C07189=1022.011,-71.493,-94.373,166.291,49.653,158.986
C07190=1022.017,-71.243,-94.384,166.295,49.649,158.986
C07191=1022.023,-70.994,-94.395,166.298,49.645,158.986
C07192=1022.028,-70.744,-94.405,166.301,49.641,158.985
C07193=1022.034,-70.494,-94.416,166.303,49.637,158.985
C07194=1022.040,-70.245,-94.427,166.306,49.634,158.985
C07195=1022.045,-69.995,-94.438,166.309,49.630,158.985
C07196=1022.051,-69.745,-94.448,166.312,49.627,158.985
C07197=1022.057,-69.465,-94.461,166.316,49.622,158.984
C07198=1022.063,-69.184,-94.472,166.319,49.618,158.984
C07199=1022.070,-68.903,-94.485,166.322,49.613,158.984
C07200=1022.076,-68.622,-94.497,166.326,49.609,158.984
C07201=1022.082,-68.373,-94.507,166.329,49.606,158.984
C07202=1022.087,-68.123,-94.518,166.332,49.601,158.983
C07203=1022.093,-67.874,-94.529,166.335,49.598,158.983
C07204=1022.099,-67.624,-94.540,166.338,49.594,158.983
C07205=1022.104,-67.374,-94.550,166.340,49.590,158.983
C07206=1022.110,-67.125,-94.561,166.343,49.587,158.983
C07207=1022.115,-66.875,-94.573,166.347,49.582,158.982
C07208=1022.121,-66.626,-94.583,166.350,49.578,158.982
C07209=1022.127,-66.376,-94.594,166.353,49.575,158.982
C07210=1022.132,-66.127,-94.605,166.356,49.571,158.982
C07211=1022.138,-65.876,-94.616,166.359,49.567,158.981
C07212=1022.144,-65.626,-94.627,166.362,49.564,158.981
C07213=1022.150,-65.377,-94.637,166.364,49.560,158.981
C07214=1022.156,-65.127,-94.648,166.368,49.555,158.981
C07215=1022.161,-64.878,-94.659,166.371,49.552,158.981
C07216=1022.166,-64.628,-94.671,166.374,49.548,158.980
C07217=1022.172,-64.378,-94.682,166.377,49.544,158.980
C07218=1022.178,-64.128,-94.693,166.379,49.540,158.980
C07219=1022.184,-63.879,-94.704,166.383,49.537,158.980
C07220=1022.190,-63.629,-94.714,166.385,49.533,158.979
C07221=1022.195,-63.379,-94.725,166.388,49.529,158.979
C07222=1022.201,-63.130,-94.736,166.392,49.525,158.979
C07223=1022.207,-62.880,-94.746,166.395,49.521,158.979
C07224=1022.213,-62.630,-94.758,166.398,49.517,158.979
C07225=1022.218,-62.380,-94.769,166.400,49.513,158.978
C07226=1022.224,-62.131,-94.780,166.404,49.510,158.978
C07227=1022.230,-61.881,-94.791,166.406,49.506,158.978
C07228=1022.236,-61.631,-94.802,166.409,49.502,158.978
C07229=1022.242,-61.382,-94.813,166.413,49.498,158.978
C07230=1022.247,-61.132,-94.824,166.416,49.494,158.977
C07231=1022.253,-60.883,-94.835,166.419,49.490,158.977
///RCONF 1,0,0,0,0,0,0,0,0,0,0,0,0,0,0,0,0,0,0,0,0,0,0,0
C07232=1022.259,-60.633,-94.846,166.421,49.486,158.977
C07233=1022.264,-60.383,-94.858,166.424,49.482,158.977
C07234=1022.270,-60.133,-94.868,166.427,49.479,158.976
C07235=1022.276,-59.884,-94.879,166.431,49.474,158.976
C07236=1022.282,-59.634,-94.890,166.434,49.470,158.976
C07237=1022.288,-59.385,-94.902,166.437,49.466,158.976
C07238=1022.294,-59.135,-94.913,166.440,49.463,158.976
C07239=1022.300,-58.886,-94.924,166.442,49.459,158.975
C07240=1022.305,-58.635,-94.936,166.445,49.455,158.975
C07241=1022.311,-58.386,-94.947,166.448,49.451,158.975
C07242=1022.317,-58.136,-94.957,166.452,49.447,158.975
C07243=1022.323,-57.887,-94.968,166.455,49.443,158.974
C07244=1022.329,-57.636,-94.980,166.458,49.439,158.974
C07245=1022.335,-57.387,-94.990,166.460,49.435,158.974
C07246=1022.340,-57.137,-95.001,166.463,49.431,158.974
C07247=1022.346,-56.888,-95.014,166.466,49.427,158.973
C07248=1022.352,-56.638,-95.025,166.470,49.424,158.973
C07249=1022.358,-56.389,-95.036,166.473,49.420,158.973
C07250=1022.364,-56.138,-95.047,166.475,49.416,158.973
C07251=1022.370,-55.889,-95.058,166.478,49.412,158.972
C07252=1022.376,-55.639,-95.069,166.481,49.408,158.972
C07253=1022.382,-55.390,-95.081,166.484,49.404,158.972
C07254=1022.387,-55.140,-95.092,166.488,49.400,158.972
C07255=1022.394,-54.890,-95.103,166.491,49.396,158.971
C07256=1022.399,-54.640,-95.114,166.493,49.392,158.971
C07257=1022.405,-54.391,-95.125,166.496,49.388,158.971
C07258=1022.412,-54.141,-95.137,166.499,49.384,158.971
C07259=1022.418,-53.892,-95.148,166.502,49.380,158.970
C07260=1022.423,-53.641,-95.160,166.505,49.376,158.970
C07261=1022.430,-53.363,-95.172,166.508,49.372,158.970
C07262=1022.437,-53.083,-95.185,166.512,49.367,158.970
C07263=1022.443,-52.803,-95.197,166.515,49.362,158.969
C07264=1022.450,-52.524,-95.210,166.518,49.358,158.969
C07265=1022.456,-52.274,-95.221,166.521,49.354,158.969
C07266=1022.462,-52.025,-95.233,166.525,49.350,158.969
C07267=1022.467,-51.775,-95.244,166.527,49.346,158.968
C07268=1022.474,-51.525,-95.256,166.530,49.342,158.968
C07269=1022.480,-51.276,-95.267,166.533,49.338,158.968
C07270=1022.485,-51.026,-95.278,166.536,49.335,158.968
C07271=1022.492,-50.776,-95.289,166.540,49.330,158.967
C07272=1022.497,-50.527,-95.302,166.543,49.326,158.967
C07273=1022.503,-50.276,-95.313,166.545,49.322,158.967
C07274=1022.509,-50.028,-95.325,166.548,49.319,158.967
C07275=1022.514,-49.777,-95.337,166.551,49.315,158.966
C07276=1022.520,-49.528,-95.348,166.554,49.312,158.966
C07277=1022.526,-49.278,-95.360,166.557,49.308,158.966
C07278=1022.532,-49.029,-95.372,166.560,49.304,158.966
C07279=1022.538,-48.778,-95.384,166.563,49.300,158.966
C07280=1022.544,-48.529,-95.395,166.566,49.296,158.965
C07281=1022.550,-48.279,-95.408,166.568,49.292,158.965
C07282=1022.555,-48.030,-95.419,166.572,49.289,158.965
C07283=1022.561,-47.780,-95.431,166.574,49.285,158.965
C07284=1022.566,-47.530,-95.443,166.577,49.281,158.964
C07285=1022.573,-47.281,-95.455,166.580,49.277,158.964
C07286=1022.578,-47.031,-95.466,166.583,49.274,158.964
C07287=1022.585,-46.781,-95.478,166.586,49.270,158.964
C07288=1022.590,-46.532,-95.490,166.588,49.266,158.963
C07289=1022.596,-46.282,-95.502,166.592,49.263,158.963
C07290=1022.601,-46.033,-95.514,166.594,49.259,158.963
C07291=1022.607,-45.783,-95.526,166.598,49.254,158.963
C07292=1022.613,-45.533,-95.537,166.601,49.251,158.963
C07293=1022.619,-45.284,-95.550,166.604,49.247,158.962
C07294=1022.625,-45.035,-95.561,166.607,49.243,158.962
C07295=1022.631,-44.784,-95.573,166.610,49.239,158.962
C07296=1022.636,-44.535,-95.585,166.613,49.236,158.962
C07297=1022.643,-44.285,-95.597,166.615,49.232,158.961
C07298=1022.648,-44.035,-95.609,166.618,49.228,158.961
C07299=1022.654,-43.786,-95.621,166.621,49.224,158.961
C07300=1022.660,-43.536,-95.633,166.624,49.221,158.961
C07301=1022.666,-43.287,-95.644,166.627,49.217,158.960
C07302=1022.672,-43.037,-95.657,166.630,49.213,158.960
C07303=1022.677,-42.788,-95.669,166.632,49.209,158.960
C07304=1022.684,-42.538,-95.681,166.635,49.205,158.960
C07305=1022.689,-42.288,-95.693,166.638,49.201,158.959
C07306=1022.695,-42.039,-95.704,166.642,49.197,158.959
C07307=1022.701,-41.789,-95.717,166.645,49.193,158.959
C07308=1022.707,-41.539,-95.729,166.648,49.189,158.958
C07309=1022.713,-41.289,-95.740,166.651,49.186,158.958
C07310=1022.719,-41.040,-95.753,166.653,49.182,158.958
C07311=1022.725,-40.791,-95.764,166.656,49.178,158.958
C07312=1022.731,-40.541,-95.777,166.659,49.174,158.957
C07313=1022.737,-40.291,-95.790,166.662,49.170,158.957
C07314=1022.743,-40.041,-95.800,166.665,49.167,158.957
C07315=1022.748,-39.792,-95.813,166.668,49.163,158.957
C07316=1022.755,-39.542,-95.825,166.670,49.159,158.956
C07317=1022.760,-39.293,-95.837,166.673,49.155,158.956
C07318=1022.766,-39.043,-95.850,166.676,49.151,158.956
C07319=1022.772,-38.793,-95.862,166.679,49.147,158.956
C07320=1022.779,-38.543,-95.874,166.682,49.143,158.955
C07321=1022.784,-38.294,-95.886,166.685,49.139,158.955
C07322=1022.790,-38.044,-95.899,166.688,49.136,158.955
C07323=1022.796,-37.794,-95.911,166.690,49.132,158.955
C07324=1022.801,-37.545,-95.923,166.693,49.128,158.954
C07325=1022.808,-37.266,-95.937,166.697,49.124,158.954
C07326=1022.815,-36.986,-95.951,166.700,49.120,158.954
C07327=1022.821,-36.708,-95.965,166.704,49.116,158.954
C07328=1022.828,-36.429,-95.979,166.706,49.112,158.953
C07329=1022.834,-36.179,-95.992,166.709,49.108,158.953
C07330=1022.839,-35.929,-96.004,166.712,49.104,158.953
C07331=1022.845,-35.680,-96.016,166.715,49.100,158.953
C07332=1022.851,-35.430,-96.028,166.718,49.096,158.952
C07333=1022.857,-35.180,-96.041,166.721,49.093,158.952
C07334=1022.863,-34.931,-96.053,166.724,49.089,158.952
C07335=1022.869,-34.681,-96.066,166.726,49.085,158.952
C07336=1022.875,-34.431,-96.078,166.729,49.081,158.951
C07337=1022.880,-34.181,-96.091,166.732,49.078,158.951
C07338=1022.886,-33.932,-96.103,166.735,49.074,158.951
C07339=1022.892,-33.682,-96.115,166.738,49.070,158.951
C07340=1022.898,-33.433,-96.127,166.741,49.066,158.950
C07341=1022.904,-33.183,-96.141,166.744,49.063,158.950
C07342=1022.910,-32.934,-96.153,166.747,49.059,158.950
C07343=1022.916,-32.684,-96.165,166.749,49.055,158.950
C07344=1022.922,-32.434,-96.178,166.752,49.051,158.949
C07345=1022.928,-32.185,-96.191,166.755,49.048,158.949
C07346=1022.933,-31.935,-96.203,166.758,49.044,158.949
C07347=1022.939,-31.686,-96.215,166.761,49.040,158.949
C07348=1022.945,-31.436,-96.229,166.764,49.036,158.948
C07349=1022.952,-31.187,-96.240,166.767,49.032,158.948
C07350=1022.958,-30.937,-96.253,166.769,49.028,158.948
C07351=1022.963,-30.687,-96.266,166.772,49.024,158.948
C07352=1022.969,-30.437,-96.278,166.775,49.020,158.947
C07353=1022.975,-30.188,-96.291,166.778,49.017,158.947
C07354=1022.981,-29.939,-96.304,166.781,49.013,158.947
C07355=1022.987,-29.689,-96.316,166.784,49.009,158.946
C07356=1022.993,-29.439,-96.329,166.786,49.005,158.946
C07357=1022.999,-29.189,-96.341,166.789,49.001,158.946
C07358=1023.006,-28.940,-96.354,166.792,48.997,158.946
C07359=1023.011,-28.690,-96.366,166.795,48.994,158.945
C07360=1023.017,-28.441,-96.379,166.798,48.990,158.945
C07361=1023.023,-28.192,-96.392,166.801,48.986,158.945
C07362=1023.029,-27.942,-96.405,166.804,48.982,158.945
C07363=1023.035,-27.692,-96.417,166.807,48.978,158.944
C07364=1023.041,-27.442,-96.430,166.810,48.974,158.944
C07365=1023.047,-27.193,-96.443,166.812,48.971,158.944
C07366=1023.053,-26.943,-96.455,166.815,48.967,158.943
C07367=1023.059,-26.694,-96.469,166.818,48.963,158.943
C07368=1023.064,-26.443,-96.482,166.821,48.960,158.943
C07369=1023.070,-26.194,-96.494,166.824,48.956,158.943
C07370=1023.076,-25.945,-96.507,166.826,48.952,158.942
C07371=1023.082,-25.695,-96.520,166.829,48.949,158.942
C07372=1023.088,-25.446,-96.533,166.832,48.945,158.942
C07373=1023.094,-25.196,-96.546,166.835,48.941,158.942
C07374=1023.099,-24.946,-96.560,166.838,48.938,158.942
C07375=1023.105,-24.696,-96.572,166.841,48.934,158.941
C07376=1023.111,-24.447,-96.585,166.844,48.930,158.941
C07377=1023.117,-24.197,-96.598,166.847,48.926,158.941
C07378=1023.123,-23.948,-96.611,166.850,48.922,158.941
C07379=1023.129,-23.698,-96.624,166.852,48.918,158.940
C07380=1023.135,-23.449,-96.638,166.854,48.915,158.940
C07381=1023.141,-23.199,-96.650,166.857,48.912,158.940
C07382=1023.147,-22.949,-96.663,166.860,48.908,158.939
C07383=1023.153,-22.700,-96.676,166.863,48.904,158.939
C07384=1023.159,-22.450,-96.689,166.866,48.900,158.939
C07385=1023.164,-22.200,-96.702,166.869,48.896,158.939
C07386=1023.170,-21.951,-96.716,166.871,48.892,158.938
C07387=1023.176,-21.701,-96.728,166.874,48.889,158.938
C07388=1023.183,-21.452,-96.742,166.877,48.885,158.938
C07389=1023.189,-21.172,-96.756,166.880,48.881,158.937
C07390=1023.196,-20.892,-96.771,166.884,48.876,158.937
C07391=1023.202,-20.612,-96.786,166.886,48.872,158.937
C07392=1023.209,-20.332,-96.800,166.890,48.867,158.937
C07393=1023.215,-20.083,-96.813,166.893,48.864,158.936
C07394=1023.221,-19.833,-96.826,166.896,48.860,158.936
C07395=1023.227,-19.582,-96.840,166.899,48.856,158.936
C07396=1023.233,-19.333,-96.853,166.901,48.852,158.935
C07397=1023.239,-19.084,-96.866,166.903,48.849,158.935
C07398=1023.245,-18.834,-96.879,166.906,48.845,158.935
C07399=1023.251,-18.585,-96.892,166.909,48.842,158.935
C07400=1023.257,-18.335,-96.906,166.912,48.838,158.934
C07401=1023.263,-18.085,-96.919,166.915,48.834,158.934
C07402=1023.269,-17.836,-96.932,166.917,48.830,158.934
C07403=1023.275,-17.587,-96.945,166.921,48.826,158.934
C07404=1023.281,-17.337,-96.958,166.923,48.822,158.933
C07405=1023.287,-17.087,-96.972,166.926,48.819,158.933
C07406=1023.293,-16.838,-96.985,166.929,48.815,158.933
C07407=1023.299,-16.588,-96.997,166.932,48.811,158.932
C07408=1023.305,-16.339,-97.011,166.934,48.807,158.932
C07409=1023.312,-16.089,-97.024,166.938,48.803,158.932
C07410=1023.317,-15.839,-97.038,166.940,48.800,158.932
C07411=1023.323,-15.589,-97.051,166.943,48.796,158.931
C07412=1023.329,-15.340,-97.064,166.946,48.792,158.931
C07413=1023.335,-15.091,-97.078,166.949,48.788,158.931
C07414=1023.341,-14.841,-97.091,166.951,48.785,158.930
C07415=1023.346,-14.592,-97.105,166.954,48.781,158.930
C07416=1023.353,-14.343,-97.118,166.956,48.777,158.930
C07417=1023.359,-14.092,-97.132,166.960,48.774,158.930
C07418=1023.365,-13.842,-97.145,166.962,48.770,158.929
C07419=1023.370,-13.593,-97.159,166.965,48.766,158.929
C07420=1023.376,-13.344,-97.172,166.968,48.763,158.929
C07421=1023.382,-13.094,-97.186,166.971,48.759,158.929
C07422=1023.388,-12.845,-97.199,166.973,48.755,158.928
C07423=1023.394,-12.595,-97.213,166.976,48.751,158.928
C07424=1023.400,-12.345,-97.227,166.979,48.748,158.928
C07425=1023.406,-12.096,-97.241,166.982,48.744,158.927
C07426=1023.412,-11.846,-97.254,166.984,48.740,158.927
C07427=1023.418,-11.597,-97.268,166.987,48.736,158.927
C07428=1023.424,-11.347,-97.281,166.990,48.733,158.927
C07429=1023.429,-11.098,-97.295,166.993,48.729,158.926
C07430=1023.436,-10.848,-97.309,166.996,48.725,158.926
C07431=1023.442,-10.598,-97.322,166.998,48.721,158.926
C07432=1023.448,-10.349,-97.336,167.001,48.718,158.925
C07433=1023.454,-10.100,-97.349,167.004,48.714,158.925
C07434=1023.459,-9.850,-97.363,167.006,48.710,158.925
C07435=1023.466,-9.600,-97.376,167.009,48.706,158.924
C07436=1023.472,-9.351,-97.390,167.012,48.703,158.924
C07437=1023.478,-9.101,-97.404,167.015,48.699,158.924
C07438=1023.483,-8.852,-97.417,167.018,48.695,158.924
C07439=1023.490,-8.602,-97.431,167.021,48.691,158.923
C07440=1023.496,-8.352,-97.445,167.022,48.687,158.923
C07441=1023.502,-8.103,-97.458,167.025,48.684,158.923
C07442=1023.507,-7.854,-97.472,167.028,48.680,158.923
C07443=1023.514,-7.604,-97.485,167.031,48.676,158.922
C07444=1023.520,-7.354,-97.500,167.034,48.672,158.922
C07445=1023.526,-7.105,-97.513,167.037,48.669,158.922
C07446=1023.531,-6.855,-97.527,167.039,48.665,158.921
C07447=1023.538,-6.605,-97.540,167.042,48.661,158.921
C07448=1023.544,-6.356,-97.555,167.045,48.657,158.921
C07449=1023.550,-6.107,-97.568,167.047,48.654,158.920
C07450=1023.556,-5.857,-97.582,167.050,48.650,158.920
C07451=1023.562,-5.607,-97.596,167.053,48.646,158.920
C07452=1023.568,-5.358,-97.610,167.056,48.642,158.919
C07453=1023.575,-5.076,-97.625,167.059,48.638,158.919
C07454=1023.582,-4.794,-97.641,167.062,48.633,158.919
C07455=1023.589,-4.513,-97.656,167.065,48.629,158.918
C07456=1023.596,-4.231,-97.671,167.069,48.625,158.918
C07457=1023.602,-3.981,-97.686,167.071,48.621,158.918
C07458=1023.607,-3.732,-97.700,167.073,48.618,158.917
C07459=1023.613,-3.483,-97.714,167.076,48.614,158.917
C07460=1023.619,-3.232,-97.728,167.079,48.610,158.917
C07461=1023.625,-2.983,-97.742,167.082,48.606,158.917
C07462=1023.631,-2.734,-97.756,167.085,48.603,158.917
C07463=1023.637,-2.484,-97.770,167.087,48.600,158.916
C07464=1023.643,-2.234,-97.784,167.090,48.596,158.916
C07465=1023.648,-1.985,-97.799,167.093,48.592,158.916
C07466=1023.654,-1.735,-97.813,167.095,48.589,158.915
C07467=1023.660,-1.486,-97.828,167.098,48.585,158.915
C07468=1023.666,-1.236,-97.842,167.100,48.582,158.915
C07469=1023.672,-0.986,-97.856,167.103,48.578,158.915
C07470=1023.678,-0.738,-97.870,167.106,48.574,158.914
C07471=1023.684,-0.488,-97.884,167.109,48.570,158.914
C07472=1023.690,-0.238,-97.899,167.112,48.567,158.914
C07473=1023.696,0.011,-97.912,167.114,48.563,158.913
C07474=1023.701,0.261,-97.926,167.116,48.559,158.913
C07475=1023.707,0.510,-97.941,167.120,48.556,158.913
C07476=1023.713,0.760,-97.955,167.122,48.552,158.913
C07477=1023.719,1.009,-97.969,167.125,48.548,158.912
C07478=1023.726,1.259,-97.983,167.127,48.545,158.912
C07479=1023.731,1.508,-97.998,167.130,48.541,158.912
C07480=1023.737,1.758,-98.012,167.133,48.537,158.911
C07481=1023.743,2.007,-98.027,167.136,48.533,158.911
C07482=1023.749,2.257,-98.041,167.139,48.530,158.911
C07483=1023.755,2.507,-98.055,167.141,48.527,158.910
C07484=1023.761,2.756,-98.069,167.143,48.523,158.910
C07485=1023.767,3.006,-98.083,167.146,48.519,158.910
C07486=1023.773,3.255,-98.098,167.149,48.515,158.909
C07487=1023.779,3.504,-98.112,167.152,48.512,158.909
C07488=1023.785,3.754,-98.126,167.154,48.508,158.909
C07489=1023.791,4.003,-98.141,167.157,48.504,158.909
C07490=1023.797,4.253,-98.155,167.160,48.500,158.908
C07491=1023.803,4.502,-98.170,167.162,48.496,158.908
C07492=1023.809,4.753,-98.184,167.166,48.493,158.908
C07493=1023.814,5.002,-98.199,167.167,48.489,158.907
C07494=1023.821,5.251,-98.212,167.170,48.486,158.907
C07495=1023.827,5.500,-98.227,167.173,48.482,158.907
C07496=1023.833,5.751,-98.241,167.176,48.478,158.906
C07497=1023.839,6.000,-98.256,167.179,48.474,158.906
C07498=1023.845,6.249,-98.271,167.182,48.471,158.906
C07499=1023.851,6.499,-98.284,167.183,48.467,158.906
C07500=1023.857,6.749,-98.299,167.186,48.463,158.905
C07501=1023.863,6.998,-98.313,167.189,48.459,158.905
C07502=1023.869,7.248,-98.328,167.192,48.455,158.905
C07503=1023.876,7.496,-98.342,167.195,48.451,158.904
C07504=1023.882,7.747,-98.356,167.197,48.449,158.904
C07505=1023.887,7.996,-98.371,167.200,48.445,158.904
C07506=1023.894,8.245,-98.386,167.202,48.441,158.903
C07507=1023.899,8.495,-98.400,167.205,48.437,158.903
C07508=1023.906,8.745,-98.415,167.208,48.433,158.903
C07509=1023.911,8.994,-98.429,167.211,48.429,158.902
C07510=1023.918,9.244,-98.444,167.213,48.425,158.902
C07511=1023.923,9.493,-98.458,167.215,48.421,158.902
C07512=1023.930,9.742,-98.473,167.218,48.418,158.901
C07513=1023.936,9.992,-98.486,167.221,48.414,158.901
C07514=1023.942,10.241,-98.501,167.224,48.410,158.901
C07515=1023.948,10.490,-98.516,167.227,48.407,158.901
C07516=1023.954,10.740,-98.531,167.229,48.403,158.900
C07517=1023.962,11.023,-98.547,167.232,48.398,158.900
C07518=1023.968,11.307,-98.564,167.235,48.394,158.899
C07519=1023.975,11.591,-98.581,167.238,48.390,158.899
C07520=1023.982,11.874,-98.597,167.242,48.385,158.899
C07521=1023.988,12.124,-98.611,167.244,48.382,158.898
C07522=1023.994,12.373,-98.626,167.247,48.378,158.898
C07523=1024.000,12.623,-98.641,167.249,48.374,158.898
C07524=1024.007,12.873,-98.656,167.252,48.370,158.897
C07525=1024.012,13.122,-98.670,167.255,48.366,158.897
C07526=1024.019,13.372,-98.684,167.257,48.362,158.897
C07527=1024.025,13.622,-98.699,167.260,48.358,158.896
C07528=1024.031,13.871,-98.714,167.262,48.356,158.896
C07529=1024.037,14.120,-98.729,167.265,48.352,158.896
C07530=1024.043,14.369,-98.743,167.268,48.348,158.895
C07531=1024.049,14.619,-98.758,167.271,48.344,158.895
C07532=1024.055,14.869,-98.774,167.273,48.340,158.895
C07533=1024.061,15.118,-98.789,167.276,48.337,158.895
C07534=1024.067,15.367,-98.803,167.278,48.333,158.894
C07535=1024.073,15.616,-98.818,167.281,48.329,158.894
C07536=1024.079,15.866,-98.833,167.284,48.325,158.894
C07537=1024.085,16.117,-98.848,167.286,48.322,158.893
C07538=1024.090,16.366,-98.862,167.289,48.319,158.893
C07539=1024.097,16.615,-98.877,167.292,48.315,158.893
C07540=1024.103,16.865,-98.892,167.295,48.311,158.892
C07541=1024.109,17.114,-98.907,167.296,48.307,158.892
C07542=1024.115,17.364,-98.922,167.299,48.303,158.892
C07543=1024.121,17.613,-98.937,167.302,48.299,158.891
C07544=1024.127,17.862,-98.952,167.305,48.296,158.891
C07545=1024.133,18.112,-98.967,167.307,48.293,158.891
C07546=1024.139,18.362,-98.982,167.310,48.289,158.890
C07547=1024.145,18.610,-98.998,167.313,48.285,158.890
C07548=1024.151,18.860,-99.013,167.316,48.281,158.890
C07549=1024.158,19.110,-99.028,167.317,48.277,158.889
C07550=1024.163,19.359,-99.042,167.320,48.274,158.889
C07551=1024.169,19.609,-99.058,167.323,48.270,158.889
C07552=1024.175,19.858,-99.073,167.326,48.266,158.888
C07553=1024.182,20.108,-99.088,167.328,48.263,158.888
C07554=1024.187,20.357,-99.103,167.331,48.259,158.888
C07555=1024.193,20.607,-99.118,167.334,48.255,158.887
C07556=1024.200,20.857,-99.133,167.336,48.251,158.887
C07557=1024.205,21.105,-99.149,167.339,48.248,158.887
C07558=1024.211,21.355,-99.164,167.341,48.244,158.886
C07559=1024.218,21.604,-99.178,167.344,48.241,158.886
C07560=1024.223,21.854,-99.194,167.347,48.237,158.886
C07561=1024.229,22.103,-99.209,167.349,48.233,158.885
C07562=1024.235,22.353,-99.224,167.352,48.229,158.885
C07563=1024.241,22.602,-99.240,167.355,48.226,158.885
C07564=1024.247,22.851,-99.254,167.358,48.222,158.885
C07565=1024.254,23.101,-99.269,167.359,48.219,158.884
C07566=1024.259,23.351,-99.285,167.362,48.215,158.884
C07567=1024.266,23.601,-99.300,167.365,48.211,158.884
C07568=1024.272,23.850,-99.316,167.368,48.207,158.883
C07569=1024.277,24.099,-99.331,167.370,48.203,158.883
C07570=1024.284,24.349,-99.346,167.373,48.200,158.883
C07571=1024.289,24.599,-99.361,167.376,48.196,158.882
C07572=1024.296,24.848,-99.377,167.378,48.192,158.882
C07573=1024.302,25.097,-99.391,167.380,48.189,158.882
C07574=1024.308,25.347,-99.407,167.383,48.185,158.881
C07575=1024.314,25.596,-99.422,167.386,48.181,158.881
C07576=1024.321,25.845,-99.438,167.389,48.177,158.881
C07577=1024.326,26.095,-99.453,167.391,48.174,158.880
C07578=1024.332,26.344,-99.468,167.394,48.170,158.880
C07579=1024.338,26.593,-99.484,167.397,48.167,158.880
C07580=1024.344,26.843,-99.499,167.398,48.163,158.879
C07581=1024.351,27.128,-99.517,167.402,48.158,158.879
C07582=1024.358,27.413,-99.534,167.405,48.154,158.878
C07583=1024.365,27.698,-99.552,167.407,48.150,158.878
C07584=1024.372,27.983,-99.570,167.411,48.146,158.878
C07585=1024.378,28.233,-99.585,167.413,48.142,158.877
C07586=1024.384,28.482,-99.601,167.416,48.138,158.877
C07587=1024.390,28.731,-99.616,167.419,48.135,158.877
C07588=1024.396,28.981,-99.631,167.421,48.131,158.876
C07589=1024.402,29.230,-99.648,167.423,48.127,158.876
C07590=1024.408,29.480,-99.663,167.426,48.124,158.876
C07591=1024.414,29.729,-99.679,167.428,48.120,158.875
C07592=1024.420,29.978,-99.693,167.431,48.117,158.875
C07593=1024.426,30.228,-99.710,167.434,48.113,158.875
C07594=1024.431,30.478,-99.725,167.436,48.109,158.874
C07595=1024.438,30.727,-99.741,167.439,48.106,158.874
C07596=1024.444,30.977,-99.756,167.442,48.102,158.874
C07597=1024.450,31.226,-99.772,167.444,48.098,158.873
C07598=1024.456,31.476,-99.788,167.447,48.095,158.873
C07599=1024.461,31.724,-99.803,167.449,48.091,158.873
C07600=1024.468,31.974,-99.818,167.452,48.087,158.872
C07601=1024.474,32.223,-99.835,167.454,48.084,158.872
C07602=1024.480,32.473,-99.850,167.457,48.080,158.872
C07603=1024.486,32.722,-99.866,167.460,48.076,158.871
C07604=1024.492,32.972,-99.882,167.462,48.072,158.871
C07605=1024.498,33.221,-99.897,167.465,48.069,158.871
C07606=1024.504,33.471,-99.913,167.467,48.065,158.870
C07607=1024.510,33.721,-99.929,167.470,48.061,158.870
C07608=1024.516,33.969,-99.944,167.472,48.058,158.870
C07609=1024.522,34.219,-99.960,167.475,48.054,158.869
C07610=1024.528,34.468,-99.975,167.478,48.050,158.869
C07611=1024.534,34.717,-99.992,167.481,48.046,158.869
C07612=1024.540,34.967,-100.007,167.482,48.043,158.868
C07613=1024.547,35.216,-100.023,167.485,48.039,158.868
C07614=1024.552,35.466,-100.038,167.488,48.035,158.868
C07615=1024.558,35.716,-100.055,167.490,48.032,158.867
C07616=1024.565,35.965,-100.070,167.493,48.028,158.867
C07617=1024.570,36.215,-100.086,167.496,48.024,158.867
C07618=1024.577,36.464,-100.101,167.499,48.021,158.866
C07619=1024.583,36.713,-100.118,167.501,48.017,158.866
C07620=1024.589,36.963,-100.133,167.503,48.013,158.866
C07621=1024.595,37.212,-100.150,167.506,48.009,158.865
C07622=1024.601,37.462,-100.166,167.508,48.006,158.865
C07623=1024.607,37.711,-100.181,167.511,48.002,158.865
C07624=1024.613,37.961,-100.197,167.514,47.999,158.864
C07625=1024.619,38.210,-100.213,167.516,47.995,158.864
C07626=1024.625,38.460,-100.230,167.519,47.991,158.864
C07627=1024.631,38.709,-100.246,167.522,47.987,158.863
C07628=1024.637,38.958,-100.262,167.523,47.984,158.863
C07629=1024.642,39.208,-100.278,167.526,47.981,158.863
C07630=1024.649,39.457,-100.293,167.529,47.977,158.862
C07631=1024.655,39.706,-100.309,167.531,47.973,158.862
C07632=1024.660,39.955,-100.325,167.534,47.969,158.862
C07633=1024.666,40.205,-100.342,167.537,47.966,158.861
C07634=1024.672,40.454,-100.358,167.539,47.962,158.861
C07635=1024.678,40.704,-100.373,167.542,47.959,158.861
C07636=1024.685,40.954,-100.390,167.545,47.955,158.860
C07637=1024.691,41.203,-100.406,167.546,47.951,158.860
C07638=1024.697,41.452,-100.422,167.549,47.948,158.860
C07639=1024.703,41.702,-100.438,167.552,47.944,158.859
C07640=1024.709,41.951,-100.454,167.554,47.940,158.859
C07641=1024.715,42.200,-100.471,167.557,47.936,158.858
C07642=1024.721,42.450,-100.487,167.560,47.932,158.858
C07643=1024.727,42.700,-100.503,167.562,47.930,158.858
C07644=1024.733,42.949,-100.519,167.565,47.926,158.857
C07645=1024.739,43.233,-100.537,167.567,47.922,158.857
C07646=1024.746,43.518,-100.556,167.570,47.917,158.857
C07647=1024.753,43.804,-100.575,167.573,47.913,158.856
C07648=1024.759,44.089,-100.594,167.577,47.909,158.856
C07649=1024.765,44.338,-100.611,167.579,47.906,158.856
C07650=1024.771,44.588,-100.627,167.581,47.902,158.855
C07651=1024.777,44.837,-100.643,167.584,47.899,158.855
C07652=1024.783,45.086,-100.659,167.586,47.895,158.855
C07653=1024.789,45.336,-100.676,167.589,47.891,158.854
C07654=1024.795,45.585,-100.692,167.591,47.888,158.854
C07655=1024.800,45.835,-100.709,167.594,47.885,158.854
C07656=1024.806,46.084,-100.725,167.596,47.881,158.853
C07657=1024.812,46.333,-100.742,167.599,47.877,158.853
C07658=1024.818,46.582,-100.758,167.602,47.873,158.853
C07659=1024.824,46.831,-100.774,167.604,47.871,158.852
C07660=1024.830,47.081,-100.791,167.607,47.867,158.852
C07661=1024.836,47.330,-100.808,167.610,47.863,158.852
C07662=1024.842,47.580,-100.824,167.611,47.859,158.851
C07663=1024.848,47.830,-100.840,167.614,47.856,158.851
C07664=1024.854,48.079,-100.857,167.616,47.853,158.851
C07665=1024.860,48.328,-100.874,167.619,47.849,158.850
C07666=1024.866,48.577,-100.890,167.622,47.845,158.850
C07667=1024.871,48.827,-100.907,167.624,47.841,158.850
C07668=1024.877,49.076,-100.923,167.627,47.838,158.849
C07669=1024.883,49.326,-100.939,167.630,47.834,158.849
C07670=1024.889,49.575,-100.955,167.632,47.831,158.849
C07671=1024.896,49.824,-100.972,167.635,47.827,158.848
C07672=1024.902,50.074,-100.989,167.637,47.823,158.848
C07673=1024.907,50.323,-101.006,167.639,47.820,158.848
C07674=1024.913,50.573,-101.022,167.642,47.816,158.847
C07675=1024.919,50.822,-101.038,167.645,47.813,158.847
C07676=1024.925,51.071,-101.055,167.647,47.809,158.847
C07677=1024.931,51.320,-101.072,167.650,47.805,158.846
C07678=1024.938,51.570,-101.088,167.652,47.802,158.846
C07679=1024.943,51.820,-101.105,167.655,47.798,158.845
C07680=1024.949,52.069,-101.122,167.657,47.794,158.845
C07681=1024.955,52.318,-101.138,167.659,47.791,158.845
C07682=1024.961,52.567,-101.155,167.662,47.787,158.844
C07683=1024.967,52.817,-101.171,167.665,47.784,158.844
C07684=1024.973,53.066,-101.189,167.667,47.780,158.844
C07685=1024.979,53.316,-101.205,167.670,47.776,158.843
C07686=1024.985,53.565,-101.221,167.673,47.772,158.843
C07687=1024.991,53.814,-101.238,167.675,47.769,158.843
C07688=1024.998,54.063,-101.255,167.678,47.765,158.842
C07689=1025.004,54.313,-101.271,167.680,47.761,158.842
C07690=1025.009,54.563,-101.288,167.682,47.758,158.842
C07691=1025.016,54.812,-101.305,167.685,47.754,158.841
C07692=1025.021,55.061,-101.321,167.688,47.750,158.841
C07693=1025.028,55.311,-101.338,167.690,47.747,158.841
C07694=1025.034,55.560,-101.355,167.693,47.743,158.840
C07695=1025.040,55.809,-101.372,167.696,47.739,158.840
C07696=1025.045,56.059,-101.388,167.698,47.736,158.840
C07697=1025.052,56.308,-101.405,167.700,47.732,158.839
C07698=1025.058,56.558,-101.422,167.703,47.728,158.839
C07699=1025.064,56.807,-101.438,167.705,47.725,158.838
C07700=1025.070,57.056,-101.455,167.708,47.721,158.838
C07701=1025.076,57.306,-101.472,167.711,47.717,158.838
C07702=1025.083,57.555,-101.489,167.714,47.713,158.837
C07703=1025.089,57.804,-101.505,167.716,47.710,158.837
C07704=1025.094,58.053,-101.521,167.718,47.706,158.837
C07705=1025.101,58.303,-101.539,167.721,47.702,158.836
C07706=1025.107,58.552,-101.556,167.723,47.699,158.836
C07707=1025.113,58.801,-101.573,167.726,47.695,158.835
C07708=1025.119,59.051,-101.589,167.729,47.691,158.835
C07709=1025.126,59.335,-101.608,167.732,47.687,158.835
C07710=1025.133,59.620,-101.628,167.734,47.683,158.834
C07711=1025.140,59.905,-101.647,167.737,47.678,158.834
C07712=1025.147,60.190,-101.666,167.741,47.674,158.833
C07713=1025.153,60.439,-101.683,167.743,47.671,158.833
C07714=1025.160,60.689,-101.700,167.745,47.667,158.833
C07715=1025.165,60.938,-101.716,167.748,47.663,158.832
C07716=1025.171,61.187,-101.734,167.750,47.659,158.832
C07717=1025.178,61.437,-101.750,167.753,47.656,158.832
C07718=1025.184,61.686,-101.767,167.756,47.652,158.831
C07719=1025.190,61.935,-101.783,167.758,47.648,158.831
C07720=1025.197,62.185,-101.801,167.761,47.644,158.830
C07721=1025.202,62.434,-101.818,167.763,47.641,158.830
C07722=1025.208,62.683,-101.835,167.766,47.637,158.830
C07723=1025.215,62.933,-101.851,167.768,47.633,158.829
C07724=1025.221,63.182,-101.868,167.771,47.629,158.829
C07725=1025.227,63.431,-101.886,167.774,47.626,158.829
C07726=1025.233,63.681,-101.902,167.776,47.622,158.828
C07727=1025.238,63.930,-101.920,167.778,47.618,158.828
C07728=1025.245,64.180,-101.937,167.781,47.614,158.828
C07729=1025.251,64.429,-101.954,167.783,47.611,158.827
C07730=1025.257,64.678,-101.971,167.786,47.607,158.827
C07731=1025.263,64.928,-101.988,167.789,47.603,158.826
C07732=1025.269,65.177,-102.005,167.791,47.600,158.826
C07733=1025.278,65.553,-102.032,167.795,47.594,158.825
C07734=1025.287,65.929,-102.057,167.799,47.589,158.825
C07735=1025.296,66.305,-102.084,167.803,47.584,158.824
C07736=1025.305,66.680,-102.109,167.806,47.578,158.824
C07737=1025.310,66.929,-102.127,167.809,47.574,158.824
C07738=1025.317,67.179,-102.144,167.811,47.571,158.823
C07739=1025.323,67.428,-102.162,167.814,47.567,158.823
C07740=1025.329,67.678,-102.178,167.817,47.563,158.822
C07741=1025.335,67.927,-102.196,167.819,47.560,158.822
C07742=1025.340,68.176,-102.214,167.821,47.556,158.822
C07743=1025.347,68.426,-102.231,167.825,47.553,158.821
C07744=1025.353,68.675,-102.248,167.826,47.549,158.821
C07745=1025.359,68.925,-102.265,167.829,47.545,158.821
C07746=1025.365,69.174,-102.283,167.832,47.542,158.820
C07747=1025.370,69.423,-102.300,167.834,47.538,158.820
C07748=1025.377,69.672,-102.318,167.837,47.534,158.820
C07749=1025.383,69.921,-102.335,167.839,47.531,158.819
C07750=1025.389,70.171,-102.353,167.842,47.528,158.819
C07751=1025.394,70.420,-102.371,167.845,47.524,158.819
C07752=1025.401,70.669,-102.388,167.847,47.520,158.818
C07753=1025.406,70.919,-102.405,167.849,47.517,158.818
C07754=1025.412,71.168,-102.422,167.852,47.513,158.817
C07755=1025.419,71.417,-102.440,167.854,47.509,158.817
C07756=1025.424,71.667,-102.457,167.857,47.506,158.817
C07757=1025.431,71.916,-102.475,167.860,47.502,158.816
C07758=1025.436,72.165,-102.493,167.862,47.499,158.816
C07759=1025.443,72.415,-102.510,167.865,47.495,158.816
C07760=1025.448,72.664,-102.528,167.867,47.492,158.815
C07761=1025.455,72.914,-102.546,167.870,47.488,158.815
C07762=1025.460,73.163,-102.563,167.873,47.484,158.815
C07763=1025.467,73.412,-102.581,167.874,47.480,158.814
C07764=1025.472,73.661,-102.598,167.877,47.477,158.814
C07765=1025.479,73.911,-102.616,167.880,47.473,158.813
C07766=1025.484,74.160,-102.634,167.882,47.469,158.813
C07767=1025.491,74.409,-102.651,167.885,47.466,158.813
C07768=1025.496,74.658,-102.669,167.888,47.462,158.812
C07769=1025.506,75.066,-102.697,167.892,47.456,158.812
C07770=1025.516,75.473,-102.726,167.895,47.451,158.811
C07771=1025.525,75.880,-102.755,167.899,47.444,158.810
C07772=1025.536,76.288,-102.784,167.904,47.439,158.810
C07773=1025.541,76.537,-102.801,167.907,47.435,158.810
C07774=1025.548,76.787,-102.819,167.909,47.431,158.809
C07775=1025.553,77.035,-102.838,167.911,47.428,158.809
C07776=1025.560,77.285,-102.856,167.914,47.424,158.809
C07777=1025.565,77.534,-102.873,167.917,47.421,158.808
C07778=1025.572,77.784,-102.890,167.919,47.417,158.808
C07779=1025.577,78.033,-102.908,167.922,47.413,158.807
C07780=1025.583,78.283,-102.927,167.924,47.410,158.807
C07781=1025.588,78.532,-102.944,167.927,47.406,158.807
C07782=1025.595,78.781,-102.963,167.930,47.403,158.807
C07783=1025.601,79.031,-102.981,167.932,47.399,158.806
C07784=1025.606,79.280,-102.998,167.935,47.396,158.806
C07785=1025.613,79.529,-103.016,167.937,47.392,158.805
C07786=1025.618,79.778,-103.035,167.939,47.388,158.805
C07787=1025.624,80.027,-103.052,167.943,47.385,158.805
C07788=1025.630,80.276,-103.070,167.945,47.382,158.804
C07789=1025.636,80.526,-103.088,167.947,47.378,158.804
C07790=1025.642,80.775,-103.106,167.949,47.374,158.804
C07791=1025.648,81.024,-103.124,167.952,47.371,158.803
C07792=1025.654,81.274,-103.142,167.955,47.367,158.803
C07793=1025.660,81.523,-103.160,167.957,47.364,158.803
C07794=1025.666,81.772,-103.178,167.960,47.360,158.802
C07795=1025.672,82.021,-103.196,167.963,47.357,158.802
C07796=1025.678,82.270,-103.215,167.965,47.353,158.801
C07797=1025.684,82.520,-103.232,167.968,47.349,158.801
C07798=1025.690,82.769,-103.250,167.970,47.346,158.801
C07799=1025.696,83.019,-103.268,167.973,47.343,158.800
C07800=1025.702,83.267,-103.286,167.976,47.339,158.800
C07801=1025.708,83.517,-103.304,167.977,47.335,158.800
C07802=1025.714,83.766,-103.323,167.980,47.332,158.799
C07803=1025.720,84.015,-103.340,167.983,47.328,158.799
C07804=1025.726,84.265,-103.358,167.985,47.324,158.799
C07805=1025.731,84.514,-103.377,167.988,47.321,158.798
C07806=1025.737,84.764,-103.395,167.991,47.317,158.798
C07807=1025.743,85.013,-103.413,167.993,47.313,158.797
C07808=1025.749,85.262,-103.431,167.996,47.310,158.797
C07809=1025.755,85.511,-103.449,167.999,47.306,158.797
C07810=1025.762,85.761,-103.468,168.001,47.303,158.796
C07811=1025.767,86.010,-103.486,168.004,47.299,158.796
C07812=1025.773,86.259,-103.503,168.006,47.295,158.796
C07813=1025.780,86.508,-103.522,168.008,47.292,158.795
C07814=1025.785,86.757,-103.540,168.011,47.288,158.795
C07815=1025.792,87.007,-103.558,168.014,47.284,158.795
C07816=1025.798,87.256,-103.576,168.016,47.281,158.794
C07817=1025.803,87.505,-103.595,168.019,47.277,158.794
C07818=1025.810,87.755,-103.612,168.022,47.273,158.793
C07819=1025.816,88.004,-103.630,168.024,47.271,158.793
C07820=1025.822,88.253,-103.649,168.027,47.267,158.793
C07821=1025.828,88.502,-103.667,168.030,47.263,158.792
C07822=1025.833,88.752,-103.686,168.032,47.259,158.792
C07823=1025.839,89.002,-103.704,168.034,47.256,158.792
C07824=1025.845,89.250,-103.722,168.037,47.252,158.791
C07825=1025.851,89.500,-103.740,168.039,47.248,158.791
C07826=1025.858,89.749,-103.759,168.042,47.245,158.790
C07827=1025.864,89.998,-103.778,168.045,47.241,158.790
C07828=1025.869,90.247,-103.795,168.047,47.238,158.790
C07829=1025.875,90.496,-103.814,168.050,47.234,158.789
C07830=1025.881,90.747,-103.833,168.052,47.231,158.789
C07831=1025.887,90.995,-103.851,168.055,47.227,158.789
C07832=1025.893,91.244,-103.870,168.058,47.223,158.788
C07833=1025.899,91.529,-103.890,168.061,47.220,158.788
C07834=1025.907,91.814,-103.912,168.063,47.216,158.788
C07835=1025.913,92.098,-103.933,168.066,47.211,158.787
C07836=1025.920,92.382,-103.954,168.069,47.208,158.787
C07837=1025.926,92.632,-103.972,168.072,47.204,158.786
C07838=1025.932,92.881,-103.992,168.074,47.200,158.786
C07839=1025.937,93.129,-104.010,168.077,47.197,158.786
C07840=1025.943,93.380,-104.028,168.080,47.194,158.785
C07841=1025.949,93.629,-104.047,168.082,47.190,158.785
C07842=1025.956,93.878,-104.066,168.085,47.186,158.785
C07843=1025.961,94.126,-104.085,168.087,47.183,158.784
C07844=1025.967,94.376,-104.103,168.089,47.179,158.784
C07845=1025.973,94.625,-104.121,168.092,47.176,158.784
C07846=1025.979,94.875,-104.140,168.095,47.172,158.783
C07847=1025.985,95.123,-104.159,168.097,47.169,158.783
C07848=1025.991,95.373,-104.177,168.100,47.165,158.782
C07849=1025.997,95.622,-104.196,168.103,47.161,158.782
C07850=1026.003,95.872,-104.215,168.105,47.158,158.782
C07851=1026.009,96.121,-104.234,168.108,47.154,158.781
C07852=1026.014,96.370,-104.251,168.111,47.151,158.781
C07853=1026.021,96.619,-104.270,168.113,47.147,158.781
C07854=1026.026,96.869,-104.289,168.116,47.144,158.780
C07855=1026.033,97.118,-104.308,168.119,47.140,158.780
C07856=1026.039,97.367,-104.327,168.121,47.136,158.779
C07857=1026.044,97.616,-104.345,168.123,47.133,158.779
C07858=1026.050,97.865,-104.363,168.126,47.129,158.779
C07859=1026.056,98.115,-104.383,168.128,47.125,158.778
C07860=1026.063,98.364,-104.401,168.131,47.122,158.778
C07861=1026.069,98.613,-104.420,168.134,47.119,158.778
C07862=1026.075,98.862,-104.439,168.136,47.115,158.777
C07863=1026.081,99.111,-104.457,168.139,47.111,158.777
C07864=1026.086,99.361,-104.476,168.142,47.108,158.777
C07865=1026.092,99.610,-104.495,168.144,47.104,158.776
C07866=1026.098,99.859,-104.514,168.147,47.100,158.776
C07867=1026.104,100.109,-104.532,168.150,47.097,158.776
C07868=1026.110,100.358,-104.552,168.152,47.094,158.775
C07869=1026.116,100.607,-104.571,168.155,47.090,158.775
C07870=1026.122,100.856,-104.589,168.158,47.086,158.774
C07871=1026.127,101.105,-104.609,168.160,47.084,158.774
C07872=1026.133,101.355,-104.628,168.163,47.080,158.774
C07873=1026.139,101.604,-104.646,168.165,47.076,158.773
C07874=1026.145,101.853,-104.666,168.167,47.073,158.773
C07875=1026.151,102.103,-104.685,168.170,47.069,158.773
C07876=1026.157,102.352,-104.704,168.173,47.066,158.772
C07877=1026.162,102.601,-104.722,168.175,47.062,158.772
C07878=1026.168,102.850,-104.742,168.178,47.059,158.772
C07879=1026.175,103.098,-104.761,168.180,47.055,158.771
C07880=1026.180,103.348,-104.780,168.183,47.052,158.771
C07881=1026.186,103.597,-104.800,168.186,47.048,158.771
C07882=1026.193,103.846,-104.818,168.188,47.045,158.770
C07883=1026.198,104.096,-104.837,168.191,47.041,158.770
C07884=1026.204,104.345,-104.857,168.194,47.037,158.770
C07885=1026.210,104.594,-104.875,168.196,47.035,158.769
C07886=1026.216,104.844,-104.895,168.199,47.031,158.769
C07887=1026.221,105.093,-104.913,168.202,47.027,158.769
C07888=1026.228,105.342,-104.932,168.204,47.024,158.768
C07889=1026.234,105.591,-104.952,168.207,47.020,158.768
C07890=1026.239,105.840,-104.971,168.210,47.017,158.768
C07891=1026.246,106.089,-104.990,168.212,47.013,158.767
C07892=1026.251,106.339,-105.009,168.215,47.010,158.767
C07893=1026.257,106.588,-105.028,168.218,47.006,158.766
C07894=1026.263,106.837,-105.047,168.220,47.002,158.766
C07895=1026.269,107.086,-105.067,168.222,46.999,158.766
C07896=1026.275,107.335,-105.086,168.226,46.996,158.765
C07897=1026.281,107.620,-105.108,168.228,46.991,158.765
C07898=1026.288,107.905,-105.130,168.231,46.988,158.764
C07899=1026.296,108.189,-105.151,168.234,46.983,158.764
C07900=1026.302,108.473,-105.174,168.238,46.979,158.764
C07901=1026.308,108.722,-105.193,168.240,46.976,158.763
C07902=1026.314,108.972,-105.212,168.243,46.972,158.763
C07903=1026.320,109.221,-105.231,168.246,46.969,158.763
C07904=1026.326,109.470,-105.251,168.249,46.965,158.762
C07905=1026.332,109.719,-105.270,168.250,46.962,158.762
C07906=1026.338,109.968,-105.289,168.253,46.958,158.761
C07907=1026.344,110.218,-105.308,168.256,46.954,158.761
C07908=1026.350,110.467,-105.328,168.258,46.951,158.761
C07909=1026.356,110.716,-105.347,168.261,46.948,158.760
C07910=1026.361,110.965,-105.366,168.264,46.944,158.760
C07911=1026.367,111.214,-105.386,168.266,46.941,158.760
C07912=1026.373,111.464,-105.405,168.269,46.937,158.759
C07913=1026.380,111.712,-105.425,168.272,46.934,158.759
C07914=1026.385,111.962,-105.444,168.274,46.930,158.759
C07915=1026.391,112.211,-105.463,168.277,46.927,158.758
C07916=1026.397,112.460,-105.483,168.280,46.923,158.758
C07917=1026.403,112.709,-105.502,168.283,46.919,158.758
C07918=1026.409,112.958,-105.522,168.285,46.916,158.757
C07919=1026.414,113.207,-105.542,168.288,46.913,158.757
C07920=1026.421,113.458,-105.561,168.290,46.910,158.757
C07921=1026.426,113.707,-105.582,168.293,46.906,158.756
C07922=1026.432,113.956,-105.602,168.296,46.902,158.756
C07923=1026.438,114.205,-105.621,168.298,46.900,158.756
C07924=1026.444,114.454,-105.641,168.301,46.896,158.755
C07925=1026.449,114.703,-105.660,168.304,46.892,158.755
C07926=1026.455,114.952,-105.680,168.306,46.889,158.755
C07927=1026.461,115.201,-105.699,168.309,46.886,158.754
C07928=1026.466,115.451,-105.720,168.312,46.882,158.754
C07929=1026.472,115.700,-105.739,168.314,46.879,158.754
C07930=1026.478,115.949,-105.759,168.317,46.875,158.753
C07931=1026.484,116.198,-105.779,168.320,46.872,158.753
C07932=1026.490,116.447,-105.798,168.322,46.869,158.753
C07933=1026.496,116.696,-105.818,168.325,46.865,158.752
C07934=1026.501,116.945,-105.838,168.328,46.862,158.752
C07935=1026.507,117.194,-105.858,168.330,46.859,158.752
C07936=1026.513,117.443,-105.878,168.333,46.855,158.751
C07937=1026.518,117.693,-105.897,168.336,46.851,158.751
C07938=1026.524,117.942,-105.917,168.338,46.849,158.751
C07939=1026.530,118.190,-105.937,168.341,46.845,158.750
C07940=1026.536,118.440,-105.957,168.344,46.841,158.750
C07941=1026.542,118.690,-105.977,168.346,46.838,158.750
C07942=1026.548,118.938,-105.997,168.349,46.835,158.749
C07943=1026.554,119.188,-106.017,168.352,46.831,158.749
C07944=1026.560,119.437,-106.037,168.355,46.828,158.749
C07945=1026.566,119.685,-106.057,168.357,46.824,158.748
C07946=1026.571,119.935,-106.076,168.360,46.821,158.748
C07947=1026.576,120.184,-106.096,168.363,46.817,158.747
C07948=1026.582,120.433,-106.116,168.365,46.814,158.747
C07949=1026.588,120.682,-106.136,168.368,46.811,158.747
C07950=1026.595,120.932,-106.156,168.371,46.807,158.746
C07951=1026.601,121.181,-106.176,168.374,46.804,158.746
C07952=1026.607,121.429,-106.196,168.376,46.800,158.746
C07953=1026.612,121.679,-106.216,168.379,46.797,158.745
C07954=1026.618,121.928,-106.236,168.382,46.794,158.745
C07955=1026.624,122.177,-106.256,168.384,46.790,158.745
C07956=1026.630,122.426,-106.276,168.387,46.786,158.744
C07957=1026.636,122.676,-106.295,168.390,46.783,158.744
C07958=1026.641,122.925,-106.316,168.393,46.780,158.744
C07959=1026.647,123.174,-106.336,168.395,46.776,158.743
C07960=1026.653,123.422,-106.356,168.398,46.773,158.743
C07961=1026.660,123.707,-106.378,168.401,46.769,158.743
C07962=1026.667,123.992,-106.402,168.405,46.765,158.742
C07963=1026.674,124.276,-106.424,168.408,46.761,158.742
C07964=1026.681,124.560,-106.447,168.411,46.757,158.741
C07965=1026.686,124.810,-106.467,168.413,46.753,158.741
C07966=1026.692,125.059,-106.487,168.417,46.750,158.741
C07967=1026.698,125.308,-106.507,168.420,46.746,158.740
C07968=1026.705,125.557,-106.527,168.421,46.743,158.740
C07969=1026.711,125.806,-106.547,168.424,46.739,158.740
C07970=1026.716,126.055,-106.568,168.428,46.736,158.739
C07971=1026.722,126.304,-106.588,168.431,46.733,158.739
C07972=1026.728,126.553,-106.607,168.432,46.729,158.739
C07973=1026.734,126.803,-106.627,168.435,46.725,158.738
C07974=1026.740,127.052,-106.647,168.439,46.722,158.738
C07975=1026.745,127.301,-106.668,168.441,46.719,158.738
C07976=1026.752,127.550,-106.688,168.444,46.715,158.737
C07977=1026.758,127.799,-106.708,168.446,46.712,158.737
C07978=1026.764,128.048,-106.728,168.450,46.709,158.737
C07979=1026.770,128.297,-106.748,168.452,46.705,158.736
C07980=1026.776,128.547,-106.769,168.455,46.701,158.736
C07981=1026.782,128.795,-106.789,168.458,46.697,158.736
C07982=1026.788,129.044,-106.809,168.460,46.694,158.735
C07983=1026.794,129.294,-106.829,168.463,46.691,158.735
C07984=1026.800,129.542,-106.849,168.466,46.687,158.734
C07985=1026.806,129.792,-106.869,168.469,46.684,158.734
C07986=1026.812,130.040,-106.889,168.472,46.680,158.734
C07987=1026.818,130.290,-106.910,168.475,46.677,158.734
C07988=1026.824,130.539,-106.930,168.477,46.673,158.733
C07989=1026.829,130.788,-106.950,168.480,46.670,158.733
C07990=1026.835,131.038,-106.971,168.483,46.667,158.733
C07991=1026.841,131.287,-106.991,168.486,46.663,158.732
C07992=1026.847,131.536,-107.012,168.488,46.660,158.732
C07993=1026.853,131.785,-107.032,168.492,46.657,158.731
C07994=1026.858,132.034,-107.053,168.494,46.653,158.731
C07995=1026.865,132.282,-107.073,168.498,46.650,158.731
C07996=1026.870,132.532,-107.094,168.500,46.647,158.730
C07997=1026.877,132.781,-107.114,168.502,46.643,158.730
C07998=1026.882,133.030,-107.135,168.506,46.640,158.730
C07999=1026.888,133.279,-107.155,168.509,46.636,158.730
C08000=1026.894,133.528,-107.176,168.511,46.633,158.729
C08001=1026.900,133.777,-107.196,168.514,46.630,158.729
C08002=1026.905,134.026,-107.217,168.517,46.626,158.728
C08003=1026.912,134.276,-107.237,168.520,46.623,158.728
C08004=1026.917,134.524,-107.258,168.523,46.619,158.728
C08005=1026.923,134.773,-107.279,168.525,46.616,158.727
C08006=1026.929,135.023,-107.299,168.528,46.613,158.727
C08007=1026.934,135.272,-107.320,168.531,46.609,158.727
C08008=1026.941,135.521,-107.341,168.534,46.606,158.727
C08009=1026.947,135.770,-107.361,168.537,46.602,158.726
C08010=1026.953,136.019,-107.381,168.539,46.599,158.726
C08011=1026.958,136.269,-107.402,168.542,46.596,158.726
C08012=1026.964,136.517,-107.424,168.545,46.592,158.725
C08013=1026.970,136.766,-107.444,168.548,46.589,158.725
C08014=1026.976,137.016,-107.464,168.551,46.586,158.725
C08015=1026.982,137.264,-107.485,168.553,46.582,158.724
C08016=1026.988,137.514,-107.506,168.556,46.579,158.724
C08017=1026.993,137.763,-107.527,168.559,46.576,158.724
C08018=1027.000,138.011,-107.547,168.562,46.572,158.723
C08019=1027.005,138.261,-107.568,168.565,46.569,158.723
C08020=1027.011,138.509,-107.589,168.568,46.565,158.723
C08021=1027.018,138.759,-107.610,168.571,46.562,158.722
C08022=1027.023,139.008,-107.630,168.574,46.559,158.722
C08023=1027.029,139.257,-107.652,168.577,46.556,158.722
C08024=1027.034,139.506,-107.673,168.580,46.552,158.721
C08025=1027.041,139.790,-107.697,168.583,46.548,158.721
C08026=1027.048,140.075,-107.721,168.586,46.545,158.721
C08027=1027.054,140.359,-107.745,168.590,46.541,158.720
C08028=1027.061,140.643,-107.768,168.592,46.537,158.720
C08029=1027.067,140.892,-107.789,168.596,46.534,158.720
C08030=1027.072,141.142,-107.810,168.599,46.530,158.719
C08031=1027.079,141.390,-107.831,168.602,46.527,158.719
C08032=1027.084,141.640,-107.852,168.604,46.524,158.719
C08033=1027.090,141.888,-107.873,168.607,46.520,158.718
C08034=1027.096,142.137,-107.895,168.610,46.517,158.718
C08035=1027.101,142.386,-107.915,168.613,46.514,158.718
C08036=1027.108,142.635,-107.936,168.616,46.511,158.718
C08037=1027.114,142.884,-107.957,168.619,46.507,158.717
C08038=1027.120,143.134,-107.978,168.621,46.504,158.717
C08039=1027.125,143.383,-107.999,168.624,46.501,158.716
C08040=1027.131,143.632,-108.020,168.627,46.498,158.716
C08041=1027.137,143.880,-108.041,168.630,46.494,158.716
C08042=1027.143,144.130,-108.062,168.634,46.491,158.716
C08043=1027.149,144.379,-108.083,168.636,46.487,158.715
C08044=1027.155,144.628,-108.105,168.639,46.484,158.715
C08045=1027.160,144.877,-108.126,168.642,46.481,158.715
C08046=1027.166,145.126,-108.147,168.645,46.477,158.714
C08047=1027.172,145.375,-108.167,168.648,46.474,158.714
C08048=1027.179,145.624,-108.189,168.651,46.471,158.714
C08049=1027.184,145.873,-108.210,168.654,46.468,158.713
C08050=1027.190,146.122,-108.231,168.657,46.464,158.713
C08051=1027.196,146.372,-108.253,168.660,46.461,158.713
C08052=1027.202,146.620,-108.274,168.662,46.458,158.712
C08053=1027.208,146.869,-108.296,168.665,46.455,158.712
C08054=1027.213,147.118,-108.316,168.668,46.451,158.712
C08055=1027.219,147.368,-108.338,168.671,46.448,158.712
C08056=1027.225,147.616,-108.359,168.674,46.444,158.711
C08057=1027.231,147.865,-108.381,168.678,46.441,158.711
C08058=1027.237,148.114,-108.402,168.681,46.438,158.711
C08059=1027.242,148.364,-108.423,168.683,46.435,158.710
C08060=1027.249,148.613,-108.444,168.686,46.432,158.710
C08061=1027.254,148.861,-108.466,168.689,46.428,158.710
C08062=1027.260,149.111,-108.487,168.692,46.425,158.710
C08063=1027.266,149.359,-108.509,168.695,46.422,158.709
C08064=1027.272,149.608,-108.530,168.698,46.419,158.709
C08065=1027.278,149.857,-108.551,168.701,46.415,158.709
C08066=1027.284,150.107,-108.572,168.704,46.412,158.708
C08067=1027.290,150.356,-108.594,168.707,46.409,158.708
C08068=1027.295,150.604,-108.615,168.710,46.406,158.708
C08069=1027.301,150.854,-108.638,168.713,46.403,158.707
C08070=1027.306,151.102,-108.659,168.716,46.399,158.707
C08071=1027.312,151.352,-108.680,168.719,46.396,158.707
C08072=1027.319,151.601,-108.702,168.722,46.392,158.706
C08073=1027.324,151.849,-108.723,168.725,46.389,158.706
C08074=1027.330,152.098,-108.745,168.728,46.386,158.706
C08075=1027.336,152.348,-108.767,168.731,46.383,158.706
C08076=1027.342,152.596,-108.788,168.735,46.380,158.705
C08077=1027.348,152.845,-108.810,168.737,46.376,158.705
C08078=1027.354,153.094,-108.831,168.740,46.373,158.705
C08079=1027.360,153.343,-108.852,168.743,46.370,158.704
C08080=1027.365,153.593,-108.875,168.746,46.367,158.704
C08081=1027.371,153.841,-108.896,168.749,46.364,158.704
C08082=1027.377,154.090,-108.918,168.752,46.360,158.704
C08083=1027.383,154.340,-108.939,168.755,46.357,158.703
C08084=1027.388,154.588,-108.961,168.759,46.354,158.703
C08085=1027.394,154.838,-108.983,168.761,46.350,158.703
C08086=1027.400,155.087,-109.004,168.765,46.347,158.703
C08087=1027.406,155.335,-109.026,168.768,46.344,158.702
C08088=1027.411,155.585,-109.048,168.770,46.341,158.702
C08089=1027.418,155.868,-109.073,168.774,46.337,158.702
C08090=1027.425,156.153,-109.098,168.777,46.334,158.701
C08091=1027.432,156.437,-109.122,168.781,46.330,158.701
C08092=1027.438,156.720,-109.148,168.784,46.327,158.701
C08093=1027.444,156.970,-109.169,168.787,46.323,158.700
C08094=1027.450,157.218,-109.190,168.790,46.320,158.700
C08095=1027.456,157.467,-109.213,168.793,46.317,158.700
C08096=1027.462,157.716,-109.235,168.796,46.313,158.699
C08097=1027.468,157.965,-109.257,168.800,46.310,158.699
C08098=1027.474,158.214,-109.278,168.803,46.307,158.699
C08099=1027.480,158.463,-109.300,168.806,46.304,158.699
C08100=1027.485,158.712,-109.323,168.809,46.301,158.698
C08101=1027.492,158.961,-109.344,168.812,46.297,158.698
C08102=1027.497,159.210,-109.365,168.815,46.294,158.698
C08103=1027.503,159.459,-109.388,168.818,46.291,158.698
C08104=1027.509,159.708,-109.410,168.822,46.288,158.697
C08105=1027.515,159.957,-109.432,168.825,46.285,158.697
C08106=1027.520,160.206,-109.455,168.827,46.282,158.697
C08107=1027.526,160.455,-109.476,168.830,46.279,158.696
C08108=1027.531,160.704,-109.499,168.833,46.276,158.696
C08109=1027.536,160.953,-109.521,168.836,46.273,158.696
C08110=1027.543,161.202,-109.543,168.840,46.270,158.696
C08111=1027.548,161.451,-109.566,168.843,46.267,158.696
C08112=1027.554,161.700,-109.588,168.846,46.264,158.695
C08113=1027.560,161.948,-109.610,168.849,46.261,158.695
C08114=1027.565,162.198,-109.632,168.852,46.257,158.695
C08115=1027.571,162.446,-109.655,168.856,46.255,158.694
C08116=1027.576,162.696,-109.677,168.858,46.252,158.694
C08117=1027.582,162.944,-109.699,168.861,46.249,158.694
C08118=1027.587,163.193,-109.722,168.864,46.246,158.694
C08119=1027.593,163.442,-109.745,168.868,46.243,158.694
C08120=1027.600,163.691,-109.767,168.871,46.240,158.693
C08121=1027.604,163.940,-109.789,168.874,46.236,158.693
C08122=1027.610,164.189,-109.812,168.877,46.233,158.693
C08123=1027.616,164.438,-109.834,168.880,46.230,158.692
C08124=1027.622,164.687,-109.856,168.883,46.227,158.692
C08125=1027.628,164.936,-109.879,168.887,46.224,158.692
C08126=1027.633,165.184,-109.901,168.890,46.221,158.692
C08127=1027.639,165.433,-109.924,168.893,46.219,158.692
C08128=1027.645,165.682,-109.946,168.896,46.216,158.691
C08129=1027.650,165.931,-109.969,168.899,46.212,158.691
C08130=1027.656,166.180,-109.992,168.903,46.209,158.691
C08131=1027.662,166.429,-110.013,168.906,46.206,158.691
C08132=1027.668,166.678,-110.036,168.909,46.203,158.690
C08133=1027.673,166.927,-110.058,168.912,46.200,158.690
C08134=1027.679,167.176,-110.080,168.915,46.197,158.690
C08135=1027.685,167.425,-110.103,168.919,46.194,158.690
C08136=1027.691,167.674,-110.126,168.922,46.191,158.689
C08137=1027.696,167.923,-110.149,168.925,46.188,158.689
C08138=1027.703,168.172,-110.171,168.928,46.185,158.689
C08139=1027.708,168.421,-110.194,168.931,46.182,158.689
C08140=1027.714,168.670,-110.216,168.935,46.179,158.688
C08141=1027.720,168.918,-110.238,168.938,46.176,158.688
C08142=1027.725,169.167,-110.261,168.941,46.173,158.688
C08143=1027.731,169.416,-110.284,168.944,46.170,158.688
C08144=1027.736,169.665,-110.306,168.947,46.166,158.687
C08145=1027.743,169.914,-110.329,168.951,46.163,158.687
C08146=1027.749,170.163,-110.352,168.954,46.160,158.687
C08147=1027.754,170.412,-110.374,168.957,46.157,158.687
C08148=1027.760,170.661,-110.397,168.960,46.154,158.686
C08149=1027.766,170.910,-110.419,168.963,46.151,158.686
C08150=1027.772,171.159,-110.442,168.967,46.148,158.686
C08151=1027.778,171.408,-110.465,168.970,46.146,158.686
C08152=1027.783,171.656,-110.488,168.973,46.143,158.685
C08153=1027.790,171.940,-110.513,168.977,46.139,158.685
C08154=1027.796,172.223,-110.539,168.980,46.135,158.685
C08155=1027.804,172.507,-110.565,168.984,46.132,158.685
C08156=1027.811,172.791,-110.590,168.988,46.128,158.684
C08157=1027.816,173.039,-110.613,168.992,46.125,158.684
C08158=1027.822,173.288,-110.636,168.995,46.122,158.684
C08159=1027.828,173.537,-110.659,168.998,46.119,158.684
C08160=1027.834,173.786,-110.682,169.001,46.116,158.683
C08161=1027.840,174.035,-110.704,169.005,46.113,158.683
C08162=1027.846,174.284,-110.727,169.008,46.110,158.683
C08163=1027.851,174.533,-110.750,169.011,46.107,158.683
C08164=1027.858,174.781,-110.773,169.014,46.104,158.682
C08165=1027.864,175.030,-110.796,169.018,46.101,158.682
C08166=1027.869,175.280,-110.818,169.021,46.098,158.682
C08167=1027.875,175.528,-110.841,169.025,46.095,158.682
C08168=1027.880,175.777,-110.864,169.028,46.092,158.681
C08169=1027.887,176.026,-110.886,169.031,46.089,158.681
C08170=1027.893,176.275,-110.909,169.034,46.086,158.681
C08171=1027.899,176.524,-110.932,169.038,46.083,158.681
C08172=1027.905,176.773,-110.955,169.041,46.080,158.680
C08173=1027.911,177.022,-110.978,169.045,46.077,158.680
C08174=1027.917,177.270,-111.001,169.048,46.073,158.680
C08175=1027.923,177.519,-111.024,169.051,46.070,158.680
C08176=1027.929,177.768,-111.047,169.055,46.067,158.679
C08177=1027.935,178.017,-111.070,169.058,46.064,158.679
C08178=1027.941,178.265,-111.093,169.061,46.061,158.679
C08179=1027.947,178.515,-111.116,169.064,46.058,158.679
C08180=1027.953,178.764,-111.139,169.069,46.055,158.679
C08181=1027.959,179.013,-111.162,169.072,46.052,158.678
C08182=1027.965,179.261,-111.184,169.075,46.049,158.678
C08183=1027.971,179.510,-111.207,169.078,46.046,158.678
C08184=1027.977,179.759,-111.230,169.082,46.043,158.678
C08185=1027.983,180.008,-111.254,169.086,46.040,158.678
C08186=1027.990,180.257,-111.276,169.089,46.037,158.677
C08187=1027.995,180.506,-111.299,169.092,46.034,158.677
C08188=1028.001,180.755,-111.322,169.095,46.031,158.677
C08189=1028.007,181.003,-111.345,169.098,46.028,158.676
C08190=1028.013,181.253,-111.369,169.103,46.025,158.676
C08191=1028.020,181.501,-111.392,169.106,46.022,158.676
C08192=1028.026,181.750,-111.415,169.109,46.019,158.676
C08193=1028.032,181.999,-111.437,169.112,46.016,158.676
C08194=1028.037,182.248,-111.460,169.116,46.013,158.675
C08195=1028.044,182.497,-111.484,169.120,46.010,158.675
C08196=1028.050,182.745,-111.507,169.123,46.007,158.675
C08197=1028.055,182.994,-111.530,169.126,46.004,158.675
C08198=1028.061,183.243,-111.554,169.130,46.001,158.674
C08199=1028.067,183.493,-111.578,169.133,45.999,158.674
C08200=1028.073,183.742,-111.601,169.136,45.996,158.674
C08201=1028.079,183.990,-111.625,169.140,45.993,158.674
C08202=1028.084,184.239,-111.648,169.144,45.990,158.674
C08203=1028.090,184.487,-111.672,169.147,45.987,158.674
C08204=1028.095,184.737,-111.696,169.151,45.984,158.673
C08205=1028.101,184.986,-111.719,169.154,45.981,158.673
C08206=1028.107,185.234,-111.743,169.157,45.979,158.673
C08207=1028.112,185.483,-111.766,169.161,45.976,158.673
C08208=1028.118,185.731,-111.790,169.164,45.973,158.673
C08209=1028.124,185.981,-111.814,169.168,45.970,158.673
C08210=1028.130,186.229,-111.838,169.171,45.967,158.672
C08211=1028.136,186.478,-111.861,169.175,45.965,158.672
C08212=1028.141,186.727,-111.885,169.178,45.962,158.672
C08213=1028.148,186.976,-111.909,169.181,45.959,158.672
C08214=1028.153,187.225,-111.932,169.185,45.957,158.672
C08215=1028.159,187.473,-111.956,169.189,45.954,158.672
C08216=1028.165,187.722,-111.980,169.192,45.951,158.671
C08217=1028.171,188.006,-112.007,169.197,45.948,158.671
C08218=1028.177,188.289,-112.034,169.200,45.945,158.671
C08219=1028.184,188.571,-112.061,169.204,45.941,158.671
C08220=1028.191,188.855,-112.089,169.209,45.938,158.671
C08221=1028.197,189.103,-112.112,169.212,45.935,158.670
C08222=1028.202,189.352,-112.136,169.215,45.932,158.670
C08223=1028.209,189.601,-112.160,169.220,45.930,158.670
C08224=1028.215,189.849,-112.183,169.223,45.927,158.670
C08225=1028.220,190.099,-112.207,169.226,45.924,158.670
C08226=1028.226,190.348,-112.231,169.230,45.922,158.670
C08227=1028.232,190.596,-112.255,169.233,45.919,158.669
C08228=1028.238,190.844,-112.279,169.237,45.916,158.669
C08229=1028.244,191.094,-112.304,169.240,45.913,158.669
C08230=1028.249,191.343,-112.327,169.244,45.911,158.669
C08231=1028.255,191.591,-112.350,169.247,45.908,158.669
C08232=1028.261,191.840,-112.375,169.251,45.904,158.668
C08233=1028.267,192.088,-112.398,169.255,45.902,158.668
C08234=1028.273,192.338,-112.423,169.258,45.899,158.668
C08235=1028.279,192.586,-112.447,169.262,45.896,158.668
C08236=1028.284,192.835,-112.470,169.266,45.894,158.668
C08237=1028.291,193.084,-112.494,169.269,45.891,158.668
C08238=1028.297,193.332,-112.518,169.272,45.888,158.667
C08239=1028.303,193.582,-112.543,169.277,45.885,158.667
C08240=1028.309,193.830,-112.566,169.280,45.883,158.667
C08241=1028.314,194.079,-112.591,169.283,45.880,158.667
C08242=1028.321,194.328,-112.615,169.288,45.877,158.667
C08243=1028.326,194.576,-112.639,169.291,45.874,158.667
C08244=1028.333,194.825,-112.663,169.295,45.872,158.667
C08245=1028.339,195.073,-112.686,169.298,45.869,158.666
C08246=1028.345,195.323,-112.711,169.302,45.866,158.666
C08247=1028.351,195.571,-112.735,169.306,45.864,158.666
C08248=1028.357,195.820,-112.759,169.309,45.861,158.666
C08249=1028.363,196.069,-112.783,169.313,45.858,158.666
C08250=1028.369,196.318,-112.808,169.317,45.855,158.666
C08251=1028.375,196.566,-112.831,169.320,45.852,158.665
C08252=1028.381,196.815,-112.856,169.324,45.849,158.665
C08253=1028.387,197.064,-112.880,169.328,45.847,158.665
C08254=1028.392,197.313,-112.904,169.332,45.844,158.665
C08255=1028.399,197.561,-112.928,169.336,45.842,158.665
C08256=1028.405,197.810,-112.952,169.339,45.839,158.665
C08257=1028.410,198.059,-112.976,169.343,45.835,158.664
C08258=1028.417,198.308,-113.000,169.347,45.833,158.664
C08259=1028.422,198.556,-113.024,169.350,45.830,158.664
C08260=1028.429,198.805,-113.049,169.354,45.828,158.664
C08261=1028.435,199.055,-113.073,169.358,45.825,158.664
C08262=1028.441,199.303,-113.097,169.362,45.822,158.664
C08263=1028.447,199.552,-113.122,169.365,45.820,158.664
C08264=1028.453,199.800,-113.146,169.369,45.817,158.663
C08265=1028.459,200.049,-113.170,169.373,45.814,158.663
C08266=1028.466,200.298,-113.194,169.376,45.811,158.663
C08267=1028.471,200.547,-113.219,169.380,45.809,158.663
C08268=1028.477,200.795,-113.244,169.384,45.806,158.663
C08269=1028.483,201.044,-113.268,169.388,45.804,158.663
C08270=1028.488,201.293,-113.293,169.391,45.801,158.663
C08271=1028.495,201.541,-113.317,169.396,45.798,158.663
C08272=1028.501,201.790,-113.342,169.399,45.796,158.662
C08273=1028.507,202.039,-113.367,169.403,45.793,158.662
C08274=1028.512,202.287,-113.392,169.407,45.790,158.662
C08275=1028.518,202.537,-113.416,169.410,45.788,158.662
C08276=1028.524,202.784,-113.441,169.415,45.785,158.662
C08277=1028.530,203.034,-113.465,169.418,45.783,158.662
C08278=1028.537,203.282,-113.490,169.422,45.781,158.662
C08279=1028.542,203.531,-113.515,169.426,45.777,158.662
C08280=1028.548,203.780,-113.539,169.429,45.775,158.662
C08281=1028.573,204.825,-113.644,169.801,45.878,158.724
C08282=1028.583,205.203,-113.684,169.805,45.876,158.724
C08283=1028.594,205.582,-113.723,169.809,45.873,158.724
C08284=1028.604,205.959,-113.762,169.814,45.870,158.724
C08285=1028.614,206.337,-113.802,169.818,45.867,158.724
C08286=1028.620,206.585,-113.828,169.821,45.866,158.724
C08287=1028.627,206.834,-113.855,169.823,45.864,158.723
C08288=1028.634,207.082,-113.881,169.826,45.862,158.723
C08289=1028.641,207.331,-113.907,169.830,45.860,158.723
C08290=1028.648,207.579,-113.933,169.832,45.859,158.723
C08291=1028.654,207.828,-113.960,169.835,45.857,158.723
C08292=1028.660,208.076,-113.986,169.838,45.855,158.723
C08293=1028.667,208.325,-114.012,169.840,45.853,158.723
C08294=1028.674,208.573,-114.038,169.844,45.852,158.723
C08295=1028.681,208.822,-114.065,169.846,45.850,158.723
C08296=1028.687,209.071,-114.091,169.849,45.848,158.723
C08297=1028.694,209.319,-114.118,169.852,45.846,158.723
C08298=1028.700,209.567,-114.144,169.855,45.845,158.723
C08299=1028.707,209.816,-114.170,169.858,45.843,158.723
C08300=1028.713,210.064,-114.197,169.861,45.841,158.723
C08301=1028.720,210.313,-114.223,169.863,45.839,158.723
C08302=1028.727,210.562,-114.250,169.866,45.838,158.723
C08303=1028.733,210.810,-114.276,169.869,45.836,158.723
C08304=1028.740,211.059,-114.303,169.872,45.834,158.723
C08305=1028.747,211.307,-114.329,169.875,45.833,158.723
C08306=1028.753,211.556,-114.357,169.877,45.831,158.722
C08307=1028.760,211.804,-114.383,169.880,45.830,158.722
C08308=1028.766,212.053,-114.410,169.884,45.827,158.722
C08309=1028.773,212.301,-114.436,169.887,45.826,158.722
C08310=1028.779,212.550,-114.463,169.889,45.825,158.722
C08311=1028.786,212.799,-114.489,169.892,45.823,158.722
C08312=1028.793,213.047,-114.515,169.896,45.821,158.722
C08313=1028.800,213.295,-114.543,169.898,45.820,158.722
C08314=1028.806,213.543,-114.569,169.901,45.818,158.722
C08315=1028.812,213.792,-114.596,169.904,45.816,158.722
C08316=1028.820,214.041,-114.622,169.906,45.815,158.722
C08317=1028.825,214.289,-114.649,169.910,45.813,158.722
C08318=1028.833,214.537,-114.676,169.913,45.811,158.722
C08319=1028.839,214.786,-114.703,169.915,45.810,158.722
C08320=1028.846,215.034,-114.729,169.918,45.808,158.722
C08321=1028.853,215.283,-114.756,169.922,45.806,158.722
C08322=1028.859,215.531,-114.783,169.924,45.805,158.722
C08323=1028.866,215.780,-114.809,169.927,45.803,158.722
C08324=1028.872,216.029,-114.836,169.930,45.802,158.722
C08325=1028.879,216.277,-114.862,169.933,45.800,158.722
C08326=1028.886,216.525,-114.890,169.936,45.798,158.722
C08327=1028.893,216.774,-114.917,169.939,45.797,158.722
C08328=1028.898,217.022,-114.943,169.941,45.795,158.722
C08329=1028.906,217.271,-114.970,169.945,45.793,158.722
C08330=1028.912,217.520,-114.997,169.948,45.792,158.722
C08331=1028.919,217.768,-115.024,169.951,45.790,158.722
C08332=1028.926,218.016,-115.050,169.953,45.788,158.722
C08333=1028.933,218.265,-115.078,169.957,45.787,158.722
C08334=1028.940,218.514,-115.104,169.960,45.785,158.722
C08335=1028.946,218.761,-115.131,169.962,45.784,158.722
C08336=1028.953,219.010,-115.158,169.966,45.782,158.722
C08337=1028.959,219.259,-115.185,169.969,45.780,158.722
C08338=1028.970,219.642,-115.227,169.973,45.778,158.722
C08339=1028.979,220.026,-115.268,169.978,45.775,158.722
C08340=1028.990,220.408,-115.310,169.982,45.774,158.722
C08341=1029.000,220.791,-115.352,169.987,45.771,158.722
C08342=1029.006,221.040,-115.379,169.990,45.770,158.722
C08343=1029.012,221.288,-115.406,169.992,45.768,158.722
C08344=1029.020,221.536,-115.433,169.996,45.767,158.722
C08345=1029.026,221.785,-115.461,169.999,45.765,158.722
C08346=1029.033,222.033,-115.488,170.002,45.763,158.722
C08347=1029.039,222.282,-115.515,170.004,45.762,158.722
C08348=1029.046,222.530,-115.542,170.008,45.760,158.722
C08349=1029.052,222.779,-115.569,170.011,45.759,158.722
C08350=1029.059,223.027,-115.597,170.014,45.758,158.722
C08351=1029.065,223.275,-115.624,170.016,45.756,158.722
C08352=1029.072,223.524,-115.651,170.020,45.755,158.722
C08353=1029.079,223.772,-115.678,170.023,45.753,158.722
C08354=1029.085,224.021,-115.705,170.025,45.751,158.722
C08355=1029.092,224.270,-115.733,170.029,45.750,158.722
C08356=1029.099,224.517,-115.760,170.032,45.748,158.722
C08357=1029.105,224.766,-115.787,170.035,45.747,158.722
C08358=1029.112,225.015,-115.815,170.038,45.745,158.722
C08359=1029.119,225.263,-115.842,170.041,45.744,158.722
C08360=1029.126,225.512,-115.869,170.044,45.743,158.722
C08361=1029.132,225.760,-115.896,170.047,45.741,158.722
C08362=1029.138,226.008,-115.924,170.051,45.740,158.722
C08363=1029.145,226.257,-115.952,170.053,45.738,158.722
C08364=1029.152,226.505,-115.978,170.056,45.737,158.722
C08365=1029.159,226.754,-116.006,170.060,45.735,158.722
C08366=1029.166,227.002,-116.033,170.062,45.733,158.722
C08367=1029.172,227.251,-116.061,170.065,45.732,158.722
C08368=1029.179,227.499,-116.088,170.069,45.731,158.722
C08369=1029.186,227.747,-116.115,170.072,45.729,158.722
C08370=1029.192,227.996,-116.143,170.074,45.728,158.722
C08371=1029.199,228.244,-116.170,170.078,45.726,158.722
C08372=1029.206,228.492,-116.198,170.081,45.725,158.722
C08373=1029.212,228.741,-116.226,170.084,45.724,158.722
C08374=1029.219,228.989,-116.254,170.087,45.723,158.722
C08375=1029.226,229.238,-116.281,170.091,45.721,158.722
C08376=1029.232,229.485,-116.309,170.093,45.720,158.722
C08377=1029.238,229.735,-116.336,170.096,45.718,158.722
C08378=1029.245,229.983,-116.363,170.100,45.717,158.722
C08379=1029.251,230.231,-116.391,170.103,45.716,158.722
C08380=1029.258,230.480,-116.419,170.105,45.714,158.723
C08381=1029.265,230.728,-116.447,170.109,45.713,158.723
C08382=1029.271,230.977,-116.474,170.112,45.711,158.723
C08383=1029.278,231.225,-116.502,170.115,45.710,158.723
C08384=1029.284,231.474,-116.530,170.119,45.709,158.723
C08385=1029.290,231.722,-116.558,170.122,45.708,158.723
C08386=1029.297,231.970,-116.586,170.124,45.706,158.723
C08387=1029.304,232.218,-116.614,170.127,45.705,158.723
C08388=1029.311,232.466,-116.642,170.131,45.703,158.723
C08389=1029.317,232.715,-116.669,170.134,45.703,158.723
C08390=1029.324,232.963,-116.697,170.137,45.701,158.723
C08391=1029.330,233.212,-116.726,170.140,45.700,158.723
C08392=1029.337,233.460,-116.753,170.143,45.698,158.723
C08393=1029.343,233.709,-116.781,170.146,45.697,158.723
C08394=1029.354,234.084,-116.823,170.151,45.695,158.723
C08395=1029.364,234.459,-116.865,170.156,45.693,158.723
C08396=1029.373,234.835,-116.908,170.160,45.691,158.724
C08397=1029.383,235.211,-116.950,170.166,45.689,158.724
C08398=1029.390,235.459,-116.978,170.169,45.688,158.724
C08399=1029.397,235.708,-117.006,170.172,45.687,158.724
C08400=1029.404,235.955,-117.034,170.175,45.685,158.724
C08401=1029.410,236.204,-117.062,170.178,45.684,158.724
C08402=1029.416,236.453,-117.090,170.181,45.683,158.724
C08403=1029.423,236.701,-117.118,170.185,45.681,158.724
C08404=1029.430,236.949,-117.146,170.188,45.680,158.724
C08405=1029.437,237.197,-117.174,170.191,45.679,158.724
C08406=1029.443,237.446,-117.202,170.195,45.678,158.724
C08407=1029.450,237.694,-117.231,170.197,45.676,158.724
C08408=1029.456,237.942,-117.258,170.200,45.675,158.724
C08409=1029.463,238.191,-117.286,170.204,45.674,158.725
C08410=1029.469,238.439,-117.315,170.207,45.673,158.725
C08411=1029.476,238.687,-117.343,170.211,45.671,158.725
C08412=1029.483,238.936,-117.371,170.213,45.670,158.725
C08413=1029.490,239.184,-117.399,170.217,45.669,158.725
C08414=1029.496,239.432,-117.427,170.220,45.667,158.725
C08415=1029.503,239.680,-117.456,170.223,45.666,158.725
C08416=1029.509,239.929,-117.484,170.226,45.665,158.725
C08417=1029.517,240.178,-117.512,170.230,45.664,158.725
C08418=1029.523,240.426,-117.541,170.233,45.663,158.725
C08419=1029.529,240.674,-117.568,170.237,45.661,158.725
C08420=1029.536,240.922,-117.597,170.239,45.660,158.725
C08421=1029.543,241.170,-117.626,170.242,45.659,158.726
C08422=1029.549,241.419,-117.654,170.246,45.658,158.726
C08423=1029.556,241.667,-117.683,170.249,45.657,158.726
C08424=1029.562,241.916,-117.711,170.252,45.656,158.726
C08425=1029.569,242.163,-117.739,170.256,45.655,158.726
C08426=1029.575,242.412,-117.768,170.259,45.653,158.726
C08427=1029.582,242.660,-117.796,170.263,45.652,158.726
C08428=1029.588,242.909,-117.826,170.266,45.651,158.726
C08429=1029.595,243.157,-117.853,170.269,45.650,158.726
C08430=1029.601,243.405,-117.882,170.273,45.649,158.727
C08431=1029.608,243.653,-117.911,170.276,45.648,158.727
C08432=1029.614,243.902,-117.939,170.278,45.647,158.727
C08433=1029.621,244.150,-117.968,170.282,45.646,158.727
C08434=1029.627,244.398,-117.997,170.285,45.644,158.727
C08435=1029.635,244.647,-118.025,170.289,45.643,158.727
C08436=1029.641,244.895,-118.054,170.292,45.642,158.727
C08437=1029.647,245.143,-118.083,170.295,45.641,158.727
C08438=1029.653,245.391,-118.112,170.299,45.640,158.728
C08439=1029.660,245.639,-118.140,170.302,45.639,158.728
C08440=1029.666,245.888,-118.169,170.305,45.638,158.728
C08441=1029.673,246.136,-118.198,170.309,45.637,158.728
C08442=1029.679,246.384,-118.227,170.312,45.636,158.728
C08443=1029.687,246.633,-118.256,170.316,45.635,158.728
C08444=1029.693,246.881,-118.285,170.318,45.634,158.728
C08445=1029.699,247.129,-118.314,170.321,45.633,158.728
C08446=1029.705,247.377,-118.343,170.326,45.632,158.729
C08447=1029.712,247.625,-118.372,170.328,45.631,158.729
C08448=1029.719,247.874,-118.400,170.331,45.630,158.729
C08449=1029.725,248.123,-118.429,170.335,45.629,158.729
C08450=1029.734,248.492,-118.472,170.340,45.627,158.729
C08451=1029.745,248.861,-118.515,170.345,45.626,158.729
C08452=1029.755,249.231,-118.558,170.350,45.624,158.730
C08453=1029.764,249.599,-118.602,170.355,45.623,158.730
C08454=1029.770,249.848,-118.630,170.359,45.622,158.730
C08455=1029.777,250.096,-118.660,170.362,45.621,158.730
C08456=1029.784,250.345,-118.689,170.365,45.620,158.730
C08457=1029.790,250.593,-118.718,170.369,45.619,158.731
C08458=1029.797,250.840,-118.747,170.372,45.618,158.731
C08459=1029.804,251.089,-118.776,170.376,45.617,158.731
C08460=1029.810,251.337,-118.805,170.379,45.616,158.731
C08461=1029.816,251.586,-118.834,170.383,45.615,158.731
C08462=1029.824,251.834,-118.863,170.386,45.614,158.731
C08463=1029.830,252.082,-118.892,170.390,45.613,158.731
C08464=1029.836,252.330,-118.921,170.393,45.612,158.732
C08465=1029.843,252.579,-118.950,170.396,45.611,158.732
C08466=1029.849,252.827,-118.979,170.400,45.610,158.732
C08467=1029.856,253.075,-119.008,170.403,45.609,158.732
C08468=1029.864,253.323,-119.038,170.407,45.608,158.732
C08469=1029.870,253.571,-119.067,170.410,45.608,158.732
C08470=1029.876,253.820,-119.096,170.414,45.607,158.733
C08471=1029.883,254.068,-119.125,170.416,45.605,158.733
C08472=1029.890,254.316,-119.154,170.420,45.604,158.733
C08473=1029.896,254.564,-119.184,170.424,45.604,158.733
C08474=1029.903,254.813,-119.213,170.428,45.603,158.733
C08475=1029.910,255.061,-119.242,170.431,45.602,158.733
C08476=1029.916,255.310,-119.272,170.434,45.600,158.733
C08477=1029.923,255.557,-119.300,170.437,45.600,158.734
C08478=1029.930,255.805,-119.330,170.441,45.599,158.734
C08479=1029.937,256.054,-119.359,170.444,45.598,158.734
C08480=1029.943,256.302,-119.388,170.449,45.597,158.734
C08481=1029.950,256.550,-119.418,170.451,45.596,158.734
C08482=1029.957,256.798,-119.447,170.455,45.595,158.735
C08483=1029.964,257.047,-119.476,170.458,45.594,158.735
C08484=1029.971,257.294,-119.506,170.462,45.593,158.735
C08485=1029.977,257.543,-119.535,170.465,45.592,158.735
C08486=1029.984,257.791,-119.564,170.470,45.591,158.735
C08487=1029.990,258.039,-119.594,170.473,45.591,158.735
C08488=1029.998,258.287,-119.623,170.476,45.589,158.736
C08489=1030.004,258.535,-119.652,170.479,45.588,158.736
C08490=1030.011,258.784,-119.682,170.483,45.587,158.736
C08491=1030.018,259.032,-119.711,170.486,45.587,158.736
C08492=1030.025,259.280,-119.741,170.490,45.586,158.736
C08493=1030.032,259.528,-119.770,170.495,45.585,158.737
C08494=1030.039,259.777,-119.799,170.498,45.584,158.737
C08495=1030.046,260.025,-119.829,170.502,45.583,158.737
C08496=1030.052,260.273,-119.858,170.505,45.582,158.737
C08497=1030.059,260.521,-119.888,170.508,45.581,158.737
C08498=1030.065,260.769,-119.917,170.511,45.580,158.737
C08499=1030.073,261.017,-119.947,170.515,45.579,158.738
C08500=1030.079,261.265,-119.976,170.519,45.578,158.738
C08501=1030.086,261.514,-120.007,170.523,45.578,158.738
C08502=1030.092,261.761,-120.036,170.526,45.577,158.738
C08503=1030.099,262.010,-120.066,170.530,45.577,158.739
C08504=1030.106,262.258,-120.096,170.534,45.576,158.739
C08505=1030.112,262.506,-120.126,170.537,45.575,158.739
C08506=1030.122,262.874,-120.171,170.542,45.574,158.739
C08507=1030.132,263.242,-120.214,170.548,45.572,158.740
C08508=1030.142,263.610,-120.258,170.553,45.572,158.740
C08509=1030.151,263.978,-120.303,170.558,45.571,158.740
C08510=1030.159,264.226,-120.333,170.563,45.570,158.741
C08511=1030.165,264.474,-120.363,170.566,45.569,158.741
C08512=1030.172,264.722,-120.393,170.570,45.568,158.741
C08513=1030.178,264.971,-120.423,170.573,45.567,158.741
C08514=1030.185,265.219,-120.453,170.577,45.567,158.741
C08515=1030.192,265.466,-120.483,170.580,45.566,158.742
C08516=1030.199,265.714,-120.513,170.584,45.565,158.742
C08517=1030.205,265.963,-120.544,170.587,45.565,158.742
C08518=1030.212,266.210,-120.573,170.591,45.564,158.742
C08519=1030.219,266.459,-120.603,170.595,45.563,158.743
C08520=1030.226,266.707,-120.634,170.598,45.563,158.743
C08521=1030.232,266.955,-120.664,170.602,45.562,158.743
C08522=1030.239,267.203,-120.694,170.606,45.561,158.743
C08523=1030.246,267.450,-120.724,170.610,45.561,158.744
C08524=1030.252,267.699,-120.755,170.613,45.560,158.744
C08525=1030.259,267.947,-120.785,170.617,45.559,158.744
C08526=1030.265,268.195,-120.815,170.621,45.559,158.744
C08527=1030.272,268.443,-120.845,170.624,45.558,158.745
C08528=1030.279,268.691,-120.875,170.628,45.557,158.745
C08529=1030.285,268.939,-120.906,170.631,45.556,158.745
C08530=1030.292,269.187,-120.936,170.636,45.556,158.745
C08531=1030.299,269.436,-120.966,170.640,45.555,158.746
C08532=1030.305,269.684,-120.996,170.643,45.554,158.746
C08533=1030.312,269.932,-121.026,170.647,45.554,158.746
C08534=1030.319,270.180,-121.057,170.650,45.553,158.746
C08535=1030.326,270.428,-121.087,170.654,45.553,158.747
C08536=1030.332,270.676,-121.118,170.658,45.552,158.747
C08537=1030.339,270.924,-121.148,170.661,45.551,158.747
C08538=1030.346,271.172,-121.179,170.666,45.551,158.747
C08539=1030.352,271.420,-121.209,170.669,45.550,158.748
C08540=1030.359,271.668,-121.240,170.673,45.550,158.748
C08541=1030.366,271.916,-121.270,170.677,45.549,158.748
C08542=1030.372,272.165,-121.301,170.680,45.549,158.749
C08543=1030.378,272.412,-121.331,170.684,45.548,158.749
C08544=1030.386,272.660,-121.362,170.688,45.548,158.749
C08545=1030.392,272.908,-121.393,170.692,45.547,158.749
C08546=1030.399,273.157,-121.423,170.696,45.547,158.750
C08547=1030.405,273.404,-121.454,170.699,45.546,158.750
C08548=1030.413,273.652,-121.484,170.703,45.546,158.750
C08549=1030.419,273.901,-121.515,170.707,45.545,158.750
C08550=1030.426,274.149,-121.546,170.711,45.545,158.751
C08551=1030.433,274.397,-121.577,170.715,45.544,158.751
C08552=1030.439,274.644,-121.608,170.718,45.544,158.751
C08553=1030.445,274.892,-121.638,170.722,45.543,158.752
C08554=1030.453,275.141,-121.668,170.727,45.542,158.752
C08555=1030.459,275.389,-121.700,170.730,45.542,158.752
C08556=1030.467,275.637,-121.730,170.734,45.541,158.753
C08557=1030.473,275.884,-121.761,170.738,45.541,158.753
C08558=1030.479,276.133,-121.792,170.741,45.540,158.753
C08559=1030.487,276.380,-121.823,170.746,45.540,158.754
C08560=1030.493,276.629,-121.853,170.750,45.539,158.754
C08561=1030.500,276.877,-121.885,170.753,45.539,158.754
C08562=1030.510,277.249,-121.930,170.759,45.538,158.755
C08563=1030.521,277.622,-121.977,170.765,45.537,158.755
C08564=1030.530,277.994,-122.024,170.771,45.537,158.756
C08565=1030.540,278.367,-122.070,170.776,45.536,158.756
C08566=1030.547,278.615,-122.102,170.780,45.536,158.756
C08567=1030.554,278.863,-122.133,170.785,45.536,158.757
C08568=1030.560,279.111,-122.164,170.788,45.535,158.757
C08569=1030.567,279.359,-122.195,170.792,45.534,158.757
C08570=1030.573,279.607,-122.227,170.796,45.534,158.758
C08571=1030.580,279.855,-122.258,170.800,45.534,158.758
C08572=1030.586,280.103,-122.289,170.804,45.533,158.758
C08573=1030.593,280.350,-122.319,170.808,45.533,158.759
C08574=1030.600,280.598,-122.351,170.811,45.533,158.759
C08575=1030.607,280.846,-122.382,170.816,45.532,158.759
C08576=1030.614,281.094,-122.414,170.820,45.532,158.760
C08577=1030.620,281.342,-122.445,170.823,45.531,158.760
C08578=1030.627,281.590,-122.476,170.827,45.531,158.760
C08579=1030.633,281.838,-122.507,170.832,45.531,158.761
C08580=1030.640,282.086,-122.539,170.835,45.531,158.761
C08581=1030.647,282.334,-122.570,170.839,45.530,158.761
C08582=1030.654,282.582,-122.602,170.844,45.530,158.762
C08583=1030.661,282.830,-122.632,170.848,45.530,158.762
C08584=1030.668,283.078,-122.664,170.851,45.529,158.762
C08585=1030.675,283.325,-122.695,170.855,45.529,158.763
C08586=1030.681,283.573,-122.727,170.860,45.528,158.763
C08587=1030.688,283.821,-122.758,170.864,45.528,158.764
C08588=1030.695,284.069,-122.790,170.867,45.528,158.764
C08589=1030.701,284.317,-122.821,170.871,45.528,158.764
C08590=1030.708,284.565,-122.852,170.876,45.527,158.765
C08591=1030.715,284.813,-122.884,170.880,45.527,158.765
C08592=1030.722,285.061,-122.915,170.883,45.527,158.765
C08593=1030.729,285.309,-122.947,170.888,45.527,158.766
C08594=1030.736,285.557,-122.979,170.892,45.526,158.766
C08595=1030.742,285.805,-123.010,170.896,45.526,158.767
C08596=1030.750,286.053,-123.041,170.899,45.525,158.767
C08597=1030.756,286.301,-123.073,170.904,45.526,158.767
C08598=1030.763,286.548,-123.105,170.908,45.525,158.768
C08599=1030.770,286.796,-123.136,170.913,45.525,158.768
C08600=1030.776,287.044,-123.168,170.916,45.525,158.768
C08601=1030.783,287.292,-123.199,170.920,45.525,158.769
C08602=1030.790,287.539,-123.231,170.924,45.524,158.769
C08603=1030.797,287.787,-123.263,170.929,45.524,158.770
C08604=1030.803,288.036,-123.295,170.932,45.524,158.770
C08605=1030.810,288.283,-123.327,170.936,45.523,158.770
C08606=1030.817,288.531,-123.359,170.941,45.523,158.771
C08607=1030.824,288.779,-123.390,170.945,45.523,158.771
C08608=1030.831,289.026,-123.422,170.950,45.523,158.772
C08609=1030.838,289.274,-123.454,170.953,45.523,158.772
C08610=1030.844,289.523,-123.486,170.957,45.523,158.772
C08611=1030.851,289.771,-123.518,170.962,45.522,158.773
C08612=1030.858,290.018,-123.550,170.966,45.522,158.773
C08613=1030.865,290.266,-123.582,170.969,45.522,158.773
C08614=1030.872,290.514,-123.613,170.974,45.522,158.774
C08615=1030.878,290.761,-123.646,170.978,45.522,158.774
C08616=1030.885,291.010,-123.678,170.982,45.522,158.775
C08617=1030.892,291.258,-123.709,170.987,45.521,158.775
C08618=1030.903,291.642,-123.759,170.993,45.521,158.776
C08619=1030.913,292.027,-123.809,171.000,45.521,158.776
C08620=1030.924,292.411,-123.859,171.006,45.521,158.777
C08621=1030.935,292.797,-123.909,171.012,45.521,158.778
C08622=1030.941,293.044,-123.941,171.016,45.521,158.778
C08623=1030.948,293.292,-123.974,171.021,45.521,158.779
C08624=1030.955,293.540,-124.005,171.025,45.521,158.779
C08625=1030.962,293.788,-124.038,171.030,45.521,158.780
C08626=1030.969,294.035,-124.070,171.034,45.520,158.780
C08627=1030.975,294.283,-124.102,171.037,45.520,158.780
C08628=1030.982,294.531,-124.135,171.042,45.521,158.781
C08629=1030.989,294.779,-124.167,171.046,45.520,158.781
C08630=1030.996,295.026,-124.200,171.051,45.521,158.782
C08631=1031.002,295.274,-124.232,171.055,45.520,158.782
C08632=1031.010,295.522,-124.265,171.060,45.521,158.783
C08633=1031.016,295.770,-124.297,171.063,45.521,158.783
C08634=1031.022,296.018,-124.330,171.068,45.521,158.784
C08635=1031.029,296.266,-124.362,171.072,45.521,158.784
C08636=1031.036,296.513,-124.395,171.076,45.521,158.785
C08637=1031.042,296.761,-124.428,171.081,45.521,158.785
C08638=1031.049,297.009,-124.461,171.085,45.521,158.786
C08639=1031.056,297.256,-124.493,171.089,45.521,158.786
C08640=1031.062,297.504,-124.526,171.093,45.521,158.786
C08641=1031.069,297.752,-124.559,171.098,45.521,158.787
C08642=1031.076,297.999,-124.591,171.102,45.522,158.788
C08643=1031.082,298.247,-124.624,171.107,45.521,158.788
C08644=1031.089,298.495,-124.657,171.111,45.522,158.789
C08645=1031.097,298.742,-124.690,171.116,45.521,158.789
C08646=1031.103,298.990,-124.722,171.119,45.522,158.789
C08647=1031.110,299.238,-124.756,171.124,45.522,158.790
C08648=1031.116,299.486,-124.788,171.128,45.522,158.790
C08649=1031.124,299.733,-124.821,171.133,45.522,158.791
C08650=1031.130,299.981,-124.854,171.137,45.522,158.791
C08651=1031.136,300.229,-124.886,171.142,45.522,158.792
C08652=1031.144,300.476,-124.920,171.146,45.522,158.792
C08653=1031.151,300.724,-124.952,171.151,45.523,158.793
C08654=1031.158,300.972,-124.985,171.155,45.523,158.794
C08655=1031.164,301.220,-125.018,171.159,45.523,158.794
C08656=1031.171,301.468,-125.051,171.163,45.523,158.794
C08657=1031.178,301.714,-125.084,171.168,45.523,158.795
C08658=1031.185,301.963,-125.117,171.172,45.524,158.796
C08659=1031.192,302.210,-125.149,171.177,45.523,158.796
C08660=1031.199,302.458,-125.183,171.181,45.524,158.796
C08661=1031.205,302.705,-125.216,171.186,45.524,158.797
C08662=1031.212,302.954,-125.249,171.190,45.524,158.798
C08663=1031.220,303.200,-125.282,171.195,45.524,158.798
C08664=1031.227,303.449,-125.315,171.199,45.524,158.799
C08665=1031.233,303.696,-125.348,171.204,45.525,158.799
C08666=1031.241,303.944,-125.381,171.208,45.525,158.800
C08667=1031.248,304.192,-125.414,171.213,45.525,158.800
C08668=1031.254,304.439,-125.448,171.218,45.525,158.801
C08669=1031.261,304.687,-125.481,171.222,45.525,158.801
C08670=1031.268,304.934,-125.513,171.226,45.525,158.802
C08671=1031.275,305.182,-125.547,171.231,45.526,158.802
C08672=1031.282,305.430,-125.580,171.236,45.526,158.803
C08673=1031.289,305.677,-125.613,171.240,45.526,158.803
C08674=1031.301,306.079,-125.667,171.247,45.527,158.804
C08675=1031.312,306.481,-125.721,171.255,45.527,158.805
C08676=1031.324,306.883,-125.775,171.262,45.527,158.806
C08677=1031.335,307.285,-125.829,171.270,45.527,158.807
C08678=1031.342,307.532,-125.861,171.274,45.528,158.807
C08679=1031.349,307.780,-125.895,171.279,45.528,158.808
C08680=1031.356,308.027,-125.929,171.283,45.528,158.808
C08681=1031.363,308.276,-125.962,171.288,45.529,158.809
C08682=1031.371,308.522,-125.995,171.293,45.529,158.810
C08683=1031.378,308.770,-126.029,171.297,45.529,158.810
C08684=1031.385,309.018,-126.062,171.302,45.530,158.811
C08685=1031.392,309.266,-126.096,171.306,45.530,158.811
C08686=1031.399,309.513,-126.129,171.311,45.530,158.812
C08687=1031.407,309.760,-126.162,171.316,45.531,158.813
C08688=1031.413,310.009,-126.196,171.320,45.531,158.813
C08689=1031.421,310.256,-126.229,171.326,45.531,158.814
C08690=1031.429,310.504,-126.263,171.330,45.532,158.814
C08691=1031.435,310.751,-126.296,171.335,45.532,158.815
C08692=1031.442,310.998,-126.330,171.340,45.532,158.815
C08693=1031.450,311.246,-126.364,171.344,45.532,158.816
C08694=1031.457,311.494,-126.398,171.349,45.533,158.816
C08695=1031.464,311.741,-126.431,171.354,45.534,158.817
C08696=1031.470,311.989,-126.465,171.358,45.534,158.818
C08697=1031.477,312.236,-126.499,171.363,45.534,158.818
C08698=1031.484,312.484,-126.533,171.368,45.535,158.819
C08699=1031.491,312.732,-126.567,171.372,45.535,158.820
C08700=1031.497,312.979,-126.601,171.377,45.536,158.820
C08701=1031.504,313.226,-126.636,171.382,45.537,158.821
C08702=1031.511,313.474,-126.670,171.386,45.537,158.821
C08703=1031.518,313.722,-126.704,171.391,45.538,158.822
C08704=1031.525,313.970,-126.738,171.396,45.538,158.823
C08705=1031.532,314.217,-126.772,171.401,45.539,158.824
C08706=1031.539,314.464,-126.806,171.406,45.539,158.824
C08707=1031.545,314.712,-126.841,171.411,45.540,158.825
C08708=1031.553,314.959,-126.874,171.415,45.540,158.825
C08709=1031.559,315.207,-126.910,171.420,45.541,158.826
C08710=1031.567,315.454,-126.943,171.425,45.541,158.827
C08711=1031.574,315.702,-126.977,171.430,45.542,158.827
C08712=1031.581,315.949,-127.012,171.434,45.543,158.828
C08713=1031.588,316.197,-127.046,171.439,45.543,158.829
C08714=1031.595,316.445,-127.080,171.444,45.544,158.829
C08715=1031.602,316.692,-127.115,171.450,45.544,158.830
C08716=1031.609,316.940,-127.149,171.454,45.545,158.831
C08717=1031.616,317.187,-127.184,171.459,45.546,158.831
C08718=1031.623,317.435,-127.218,171.464,45.546,158.832
C08719=1031.630,317.682,-127.252,171.468,45.547,158.833
C08720=1031.637,317.930,-127.287,171.473,45.548,158.833
C08721=1031.644,318.177,-127.321,171.478,45.548,158.834
C08722=1031.651,318.425,-127.356,171.484,45.549,158.835
C08723=1031.658,318.672,-127.390,171.489,45.549,158.835
C08724=1031.666,318.920,-127.424,171.493,45.550,158.836
C08725=1031.672,319.167,-127.459,171.498,45.551,158.837
C08726=1031.680,319.415,-127.493,171.503,45.552,158.837
C08727=1031.686,319.662,-127.528,171.507,45.552,158.838
C08728=1031.694,319.909,-127.563,171.513,45.552,158.839
C08729=1031.700,320.157,-127.597,171.518,45.553,158.839
C08730=1031.713,320.564,-127.654,171.526,45.554,158.840
C08731=1031.724,320.971,-127.711,171.535,45.556,158.842
C08732=1031.736,321.377,-127.768,171.543,45.556,158.843
C08733=1031.748,321.784,-127.825,171.551,45.558,158.844
C08734=1031.755,322.032,-127.859,171.556,45.559,158.845
C08735=1031.762,322.279,-127.894,171.561,45.560,158.845
C08736=1031.770,322.527,-127.929,171.566,45.560,158.846
C08737=1031.778,322.774,-127.964,171.570,45.561,158.847
C08738=1031.784,323.021,-127.999,171.576,45.561,158.847
C08739=1031.792,323.268,-128.033,171.581,45.562,158.848
C08740=1031.798,323.516,-128.068,171.586,45.563,158.849
C08741=1031.806,323.764,-128.103,171.592,45.564,158.850
C08742=1031.813,324.011,-128.138,171.597,45.565,158.850
C08743=1031.821,324.258,-128.172,171.601,45.565,158.851
C08744=1031.828,324.506,-128.208,171.606,45.566,158.852
C08745=1031.836,324.753,-128.242,171.612,45.566,158.853
C08746=1031.843,325.000,-128.277,171.617,45.567,158.853
C08747=1031.850,325.249,-128.312,171.622,45.568,158.854
C08748=1031.858,325.496,-128.347,171.627,45.569,158.855
C08749=1031.865,325.743,-128.382,171.632,45.570,158.855
C08750=1031.873,325.991,-128.417,171.637,45.571,158.856
C08751=1031.880,326.238,-128.452,171.643,45.571,158.857
C08752=1031.887,326.485,-128.487,171.648,45.572,158.858
C08753=1031.894,326.733,-128.522,171.653,45.573,158.858
C08754=1031.902,326.980,-128.557,171.659,45.574,158.859
C08755=1031.909,327.228,-128.592,171.663,45.575,158.860
C08756=1031.917,327.475,-128.627,171.668,45.575,158.861
C08757=1031.925,327.723,-128.663,171.674,45.576,158.861
C08758=1031.932,327.970,-128.697,171.679,45.577,158.862
C08759=1031.939,328.217,-128.733,171.684,45.578,158.863
C08760=1031.946,328.465,-128.768,171.690,45.579,158.864
C08761=1031.953,328.712,-128.804,171.695,45.580,158.865
C08762=1031.961,328.960,-128.839,171.700,45.581,158.865
C08763=1031.968,329.207,-128.875,171.706,45.582,158.866
C08764=1031.976,329.455,-128.910,171.711,45.583,158.867
C08765=1031.983,329.702,-128.945,171.716,45.584,158.868
C08766=1031.990,329.949,-128.981,171.722,45.585,158.869
C08767=1031.997,330.197,-129.017,171.727,45.586,158.869
C08768=1032.004,330.444,-129.053,171.731,45.587,158.870
C08769=1032.011,330.692,-129.088,171.738,45.588,158.871
C08770=1032.019,330.938,-129.124,171.742,45.589,158.872
C08771=1032.027,331.185,-129.159,171.747,45.590,158.873
C08772=1032.034,331.433,-129.195,171.753,45.591,158.874
C08773=1032.041,331.680,-129.231,171.758,45.592,158.874
C08774=1032.049,331.928,-129.266,171.764,45.593,158.875
C08775=1032.056,332.175,-129.302,171.769,45.594,158.876
C08776=1032.064,332.423,-129.338,171.774,45.596,158.877
C08777=1032.070,332.670,-129.374,171.780,45.596,158.878
C08778=1032.078,332.917,-129.410,171.785,45.598,158.879
C08779=1032.085,333.164,-129.446,171.791,45.598,158.879
C08780=1032.092,333.412,-129.481,171.796,45.600,158.880
C08781=1032.100,333.660,-129.517,171.802,45.600,158.881
C08782=1032.108,333.906,-129.553,171.807,45.602,158.882
C08783=1032.116,334.153,-129.589,171.812,45.603,158.883
C08784=1032.123,334.402,-129.624,171.818,45.604,158.884
C08785=1032.130,334.648,-129.660,171.823,45.605,158.884
C08786=1032.142,335.050,-129.720,171.833,45.607,158.886
C08787=1032.153,335.453,-129.778,171.842,45.609,158.887
C08788=1032.165,335.855,-129.837,171.850,45.611,158.889
C08789=1032.178,336.257,-129.896,171.859,45.613,158.890
C08790=1032.185,336.504,-129.932,171.865,45.614,158.891
C08791=1032.193,336.752,-129.968,171.870,45.615,158.892
C08792=1032.200,336.999,-130.004,171.876,45.616,158.893
C08793=1032.207,337.246,-130.041,171.881,45.618,158.894
C08794=1032.215,337.494,-130.077,171.888,45.619,158.895
C08795=1032.222,337.741,-130.114,171.893,45.621,158.896
C08796=1032.230,337.987,-130.150,171.899,45.622,158.897
C08797=1032.237,338.235,-130.186,171.904,45.623,158.897
C08798=1032.245,338.482,-130.223,171.910,45.624,158.898
C08799=1032.252,338.730,-130.259,171.915,45.625,158.899
C08800=1032.260,338.977,-130.296,171.921,45.627,158.900
C08801=1032.267,339.224,-130.332,171.926,45.628,158.901
C08802=1032.275,339.471,-130.368,171.932,45.629,158.902
C08803=1032.282,339.718,-130.405,171.937,45.631,158.903
C08804=1032.289,339.966,-130.441,171.944,45.632,158.904
C08805=1032.297,340.213,-130.478,171.950,45.633,158.905
C08806=1032.305,340.460,-130.515,171.955,45.635,158.906
C08807=1032.313,340.707,-130.551,171.961,45.636,158.907
C08808=1032.320,340.955,-130.588,171.966,45.637,158.908
C08809=1032.328,341.203,-130.625,171.972,45.639,158.908
C08810=1032.335,341.449,-130.661,171.977,45.640,158.909
C08811=1032.342,341.696,-130.698,171.984,45.641,158.910
C08812=1032.350,341.943,-130.735,171.990,45.643,158.911
C08813=1032.357,342.190,-130.772,171.995,45.645,158.912
C08814=1032.365,342.438,-130.809,172.001,45.646,158.913
C08815=1032.373,342.685,-130.845,172.006,45.647,158.914
C08816=1032.380,342.932,-130.882,172.013,45.648,158.915
C08817=1032.388,343.179,-130.919,172.019,45.650,158.916
C08818=1032.395,343.426,-130.957,172.024,45.652,158.917
C08819=1032.403,343.674,-130.993,172.030,45.653,158.918
C08820=1032.410,343.921,-131.031,172.036,45.655,158.919
C08821=1032.418,344.168,-131.067,172.042,45.656,158.920
C08822=1032.426,344.415,-131.104,172.048,45.657,158.921
C08823=1032.433,344.662,-131.141,172.053,45.660,158.922
C08824=1032.441,344.909,-131.178,172.059,45.661,158.923
C08825=1032.448,345.156,-131.216,172.066,45.662,158.924
C08826=1032.455,345.403,-131.253,172.071,45.664,158.925
C08827=1032.463,345.650,-131.290,172.077,45.665,158.926
C08828=1032.471,345.898,-131.328,172.084,45.667,158.927
C08829=1032.479,346.145,-131.365,172.089,45.668,158.928
C08830=1032.486,346.392,-131.402,172.095,45.670,158.929
C08831=1032.494,346.639,-131.439,172.101,45.671,158.930
C08832=1032.502,346.886,-131.477,172.107,45.674,158.931
C08833=1032.510,347.133,-131.514,172.113,45.675,158.932
C08834=1032.517,347.380,-131.551,172.119,45.677,158.934
C08835=1032.525,347.627,-131.589,172.125,45.678,158.934
C08836=1032.533,347.875,-131.626,172.131,45.680,158.936
C08837=1032.541,348.121,-131.663,172.137,45.681,158.937
C08838=1032.548,348.369,-131.701,172.143,45.683,158.938
C08839=1032.556,348.616,-131.738,172.149,45.685,158.939
C08840=1032.564,348.863,-131.775,172.155,45.686,158.940
C08841=1032.571,349.110,-131.814,172.161,45.688,158.941
C08842=1032.584,349.509,-131.875,172.172,45.691,158.943
C08843=1032.596,349.907,-131.935,172.181,45.693,158.944
C08844=1032.608,350.307,-131.996,172.191,45.696,158.946
C08845=1032.621,350.706,-132.057,172.201,45.699,158.948
C08846=1032.628,350.953,-132.095,172.207,45.701,158.949
C08847=1032.636,351.199,-132.132,172.213,45.703,158.950
C08848=1032.644,351.447,-132.170,172.219,45.705,158.951
C08849=1032.652,351.693,-132.208,172.226,45.707,158.952
C08850=1032.659,351.941,-132.246,172.232,45.708,158.953
C08851=1032.667,352.188,-132.285,172.238,45.709,158.954
C08852=1032.675,352.435,-132.322,172.244,45.712,158.956
C08853=1032.683,352.681,-132.360,172.250,45.713,158.957
C08854=1032.691,352.929,-132.398,172.257,45.715,158.958
C08855=1032.698,353.175,-132.436,172.263,45.717,158.959
C08856=1032.706,353.423,-132.475,172.269,45.719,158.960
C08857=1032.714,353.669,-132.511,172.276,45.720,158.961
C08858=1032.722,353.917,-132.550,172.282,45.723,158.963
C08859=1032.730,354.163,-132.588,172.288,45.725,158.964
C08860=1032.738,354.410,-132.627,172.294,45.727,158.965
C08861=1032.745,354.658,-132.664,172.301,45.728,158.966
C08862=1032.754,354.904,-132.702,172.307,45.730,158.967
C08863=1032.762,355.151,-132.741,172.314,45.732,158.968
C08864=1032.770,355.398,-132.779,172.320,45.734,158.969
C08865=1032.778,355.645,-132.818,172.327,45.736,158.971
C08866=1032.785,355.893,-132.855,172.333,45.738,158.972
C08867=1032.793,356.139,-132.894,172.340,45.740,158.973
C08868=1032.801,356.386,-132.932,172.345,45.742,158.974
C08869=1032.809,356.633,-132.971,172.352,45.744,158.975
C08870=1032.817,356.880,-133.009,172.358,45.746,158.976
C08871=1032.824,357.127,-133.047,172.365,45.748,158.978
C08872=1032.833,357.373,-133.087,172.371,45.750,158.979
C08873=1032.841,357.620,-133.125,172.378,45.752,158.980
C08874=1032.849,357.867,-133.164,172.384,45.754,158.981
C08875=1032.857,358.114,-133.202,172.391,45.756,158.983
C08876=1032.865,358.361,-133.241,172.398,45.758,158.984
C08877=1032.872,358.608,-133.279,172.404,45.760,158.985
C08878=1032.881,358.855,-133.318,172.411,45.763,158.986
C08879=1032.889,359.102,-133.357,172.417,45.764,158.987
C08880=1032.897,359.348,-133.395,172.424,45.767,158.989
C08881=1032.905,359.595,-133.434,172.430,45.769,158.990
C08882=1032.913,359.842,-133.473,172.437,45.771,158.991
C08883=1032.921,360.089,-133.512,172.443,45.773,158.992
C08884=1032.928,360.336,-133.551,172.450,45.775,158.994
C08885=1032.937,360.583,-133.590,172.457,45.777,158.995
C08886=1032.945,360.830,-133.629,172.463,45.779,158.996
C08887=1032.953,361.076,-133.668,172.470,45.782,158.998
C08888=1032.961,361.323,-133.706,172.478,45.784,158.999
C08889=1032.969,361.569,-133.745,172.484,45.786,159.000
C08890=1032.977,361.817,-133.785,172.491,45.788,159.002
C08891=1032.985,362.064,-133.824,172.498,45.790,159.003
C08892=1032.993,362.311,-133.863,172.504,45.792,159.004
C08893=1033.000,362.557,-133.902,172.511,45.795,159.005
C08894=1033.009,362.804,-133.941,172.518,45.797,159.007
C08895=1033.017,363.050,-133.981,172.524,45.800,159.008
C08896=1033.025,363.298,-134.020,172.531,45.802,159.009
C08897=1033.033,363.544,-134.059,172.538,45.804,159.011
C08898=1033.046,363.950,-134.124,172.550,45.808,159.013
C08899=1033.060,364.355,-134.188,172.561,45.812,159.015
C08900=1033.073,364.759,-134.254,172.572,45.816,159.017
C08901=1033.087,365.164,-134.318,172.583,45.820,159.019
C08902=1033.094,365.411,-134.358,172.590,45.822,159.021
C08903=1033.103,365.658,-134.397,172.597,45.824,159.022
C08904=1033.111,365.905,-134.437,172.604,45.827,159.023
C08905=1033.119,366.151,-134.477,172.611,45.829,159.025
C08906=1033.127,366.398,-134.516,172.618,45.832,159.026
C08907=1033.136,366.645,-134.555,172.625,45.834,159.028
C08908=1033.144,366.892,-134.595,172.632,45.836,159.029
C08909=1033.152,367.138,-134.634,172.639,45.839,159.030
C08910=1033.160,367.385,-134.674,172.646,45.842,159.032
C08911=1033.168,367.631,-134.714,172.653,45.844,159.033
C08912=1033.177,367.878,-134.754,172.661,45.846,159.035
C08913=1033.185,368.125,-134.794,172.668,45.849,159.036
C08914=1033.194,368.372,-134.833,172.674,45.851,159.037
C08915=1033.202,368.618,-134.873,172.681,45.854,159.039
C08916=1033.210,368.865,-134.913,172.689,45.856,159.040
C08917=1033.219,369.111,-134.953,172.696,45.859,159.042
C08918=1033.227,369.358,-134.994,172.703,45.861,159.043
C08919=1033.236,369.605,-135.033,172.711,45.864,159.044
C08920=1033.243,369.852,-135.073,172.718,45.866,159.046
C08921=1033.252,370.098,-135.113,172.725,45.869,159.047
C08922=1033.260,370.344,-135.154,172.732,45.871,159.049
C08923=1033.269,370.592,-135.194,172.739,45.874,159.050
C08924=1033.277,370.838,-135.234,172.746,45.877,159.052
C08925=1033.285,371.085,-135.274,172.754,45.879,159.053
C08926=1033.293,371.331,-135.314,172.761,45.882,159.055
C08927=1033.302,371.577,-135.355,172.768,45.885,159.056
C08928=1033.310,371.824,-135.395,172.776,45.888,159.058
C08929=1033.318,372.071,-135.435,172.783,45.891,159.059
C08930=1033.326,372.317,-135.476,172.790,45.893,159.061
C08931=1033.336,372.564,-135.516,172.798,45.896,159.062
C08932=1033.344,372.810,-135.557,172.805,45.899,159.064
C08933=1033.352,373.057,-135.598,172.813,45.901,159.065
C08934=1033.361,373.303,-135.638,172.820,45.904,159.067
C08935=1033.369,373.550,-135.678,172.828,45.907,159.068
C08936=1033.377,373.797,-135.719,172.835,45.910,159.070
C08937=1033.385,374.043,-135.760,172.842,45.913,159.071
C08938=1033.395,374.290,-135.800,172.850,45.915,159.073
C08939=1033.403,374.536,-135.841,172.857,45.918,159.074
C08940=1033.411,374.782,-135.881,172.865,45.921,159.076
C08941=1033.420,375.028,-135.922,172.872,45.924,159.078
C08942=1033.428,375.275,-135.963,172.880,45.926,159.079
C08943=1033.437,375.522,-136.004,172.887,45.930,159.081
C08944=1033.446,375.769,-136.045,172.895,45.932,159.082
C08945=1033.454,376.015,-136.085,172.902,45.935,159.084
C08946=1033.463,376.262,-136.126,172.911,45.938,159.085
C08947=1033.471,376.507,-136.168,172.919,45.941,159.087
C08948=1033.480,376.754,-136.209,172.926,45.944,159.089
C08949=1033.489,377.000,-136.249,172.934,45.947,159.090
C08950=1033.497,377.247,-136.290,172.941,45.950,159.092
C08951=1033.506,377.494,-136.331,172.949,45.953,159.094
C08952=1033.514,377.740,-136.372,172.957,45.955,159.095
C08953=1033.524,377.986,-136.413,172.964,45.958,159.097
C08954=1033.531,378.199,-136.449,172.971,45.961,159.098
C08955=1033.539,378.412,-136.484,172.978,45.963,159.100
C08956=1033.545,378.625,-136.520,172.985,45.966,159.101
C08957=1033.553,378.838,-136.556,172.991,45.970,159.103
C08958=1033.561,379.051,-136.592,172.998,45.972,159.104
C08959=1033.568,379.264,-136.628,173.005,45.975,159.105
C08960=1033.575,379.477,-136.663,173.012,45.977,159.107
C08961=1033.583,379.690,-136.699,173.019,45.980,159.108
C08962=1033.591,379.937,-136.741,173.027,45.983,159.110
C08963=1033.600,380.182,-136.782,173.034,45.986,159.111
C08964=1033.609,380.429,-136.824,173.042,45.989,159.113
C08965=1033.618,380.675,-136.865,173.051,45.992,159.115
C08966=1033.627,380.921,-136.907,173.058,45.996,159.117
C08967=1033.635,381.168,-136.948,173.066,45.999,159.118
C08968=1033.644,381.414,-136.989,173.075,46.002,159.120
C08969=1033.653,381.660,-137.031,173.083,46.005,159.122
C08970=1033.661,381.907,-137.073,173.090,46.008,159.123
C08971=1033.670,382.153,-137.115,173.098,46.011,159.125
C08972=1033.679,382.400,-137.157,173.107,46.015,159.127
C08973=1033.688,382.646,-137.199,173.115,46.018,159.129
C08974=1033.696,382.893,-137.240,173.122,46.021,159.130
C08975=1033.706,383.138,-137.283,173.131,46.024,159.132
C08976=1033.715,383.385,-137.325,173.139,46.028,159.134
C08977=1033.724,383.631,-137.366,173.147,46.031,159.136
C08978=1033.732,383.877,-137.408,173.156,46.034,159.138
C08979=1033.741,384.124,-137.450,173.163,46.038,159.139
C08980=1033.751,384.369,-137.492,173.171,46.041,159.141
C08981=1033.760,384.616,-137.534,173.180,46.044,159.143
C08982=1033.769,384.862,-137.576,173.188,46.047,159.145
C08983=1033.777,385.108,-137.619,173.197,46.051,159.147
C08984=1033.786,385.355,-137.660,173.205,46.054,159.148
C08985=1033.795,385.601,-137.702,173.213,46.057,159.150
C08986=1033.804,385.847,-137.744,173.222,46.061,159.152
C08987=1033.813,386.093,-137.786,173.230,46.064,159.154
C08988=1033.822,386.339,-137.829,173.239,46.068,159.156
